C09134=1209.078,130.701,-51.461,-178.311,5.912,148.550
C09135=1209.083,130.452,-51.442,-178.314,5.911,148.551
C09136=1209.088,130.204,-51.422,-178.316,5.909,148.551
C09137=1209.093,129.954,-51.402,-178.318,5.908,148.552
C09138=1209.097,129.705,-51.382,-178.322,5.907,148.552
C09139=1209.102,129.455,-51.362,-178.324,5.906,148.553
C09140=1209.106,129.206,-51.342,-178.327,5.904,148.553
C09141=1209.112,128.957,-51.322,-178.329,5.904,148.554
C09142=1209.117,128.708,-51.301,-178.332,5.902,148.554
C09143=1209.121,128.459,-51.282,-178.334,5.901,148.555
C09144=1209.126,128.210,-51.261,-178.337,5.899,148.555
C09145=1209.131,127.960,-51.242,-178.340,5.899,148.556
C09146=1209.135,127.711,-51.221,-178.342,5.897,148.556
C09147=1209.140,127.462,-51.202,-178.345,5.896,148.557
C09148=1209.145,127.213,-51.182,-178.348,5.895,148.557
C09149=1209.150,126.964,-51.162,-178.350,5.894,148.558
C09150=1209.154,126.715,-51.142,-178.353,5.892,148.558
C09151=1209.159,126.466,-51.122,-178.355,5.891,148.559
C09152=1209.164,126.217,-51.102,-178.358,5.890,148.559
C09153=1209.169,125.968,-51.082,-178.360,5.889,148.560
C09154=1209.173,125.718,-51.063,-178.363,5.888,148.560
C09155=1209.178,125.469,-51.042,-178.366,5.886,148.561
C09156=1209.183,125.220,-51.023,-178.368,5.885,148.561
C09157=1209.188,124.971,-51.003,-178.371,5.884,148.562
C09158=1209.192,124.722,-50.983,-178.373,5.883,148.562
C09159=1209.197,124.472,-50.963,-178.376,5.882,148.563
C09160=1209.202,124.224,-50.943,-178.378,5.881,148.563
C09161=1209.207,123.974,-50.924,-178.381,5.879,148.564
C09162=1209.211,123.725,-50.904,-178.384,5.878,148.564
C09163=1209.216,123.476,-50.884,-178.386,5.877,148.565
C09164=1209.221,123.227,-50.864,-178.389,5.876,148.565
C09165=1209.226,122.977,-50.845,-178.392,5.874,148.566
C09166=1209.231,122.728,-50.825,-178.394,5.874,148.566
C09167=1209.236,122.480,-50.805,-178.396,5.873,148.567
C09168=1209.241,122.230,-50.785,-178.399,5.871,148.567
C09169=1209.245,121.980,-50.766,-178.402,5.870,148.568
C09170=1209.250,121.731,-50.746,-178.405,5.869,148.568
C09171=1209.254,121.483,-50.727,-178.407,5.868,148.569
C09172=1209.259,121.233,-50.707,-178.410,5.866,148.569
C09173=1209.264,120.984,-50.687,-178.412,5.865,148.570
C09174=1209.269,120.735,-50.668,-178.415,5.864,148.570
C09175=1209.274,120.485,-50.648,-178.417,5.863,148.571
C09176=1209.278,120.236,-50.628,-178.420,5.862,148.571
C09177=1209.284,119.988,-50.609,-178.423,5.861,148.572
C09178=1209.288,119.738,-50.589,-178.425,5.860,148.572
C09179=1209.292,119.489,-50.570,-178.428,5.858,148.573
C09180=1209.298,119.240,-50.551,-178.430,5.857,148.573
C09181=1209.303,118.990,-50.531,-178.433,5.856,148.574
C09182=1209.307,118.741,-50.511,-178.436,5.855,148.574
C09183=1209.312,118.492,-50.491,-178.438,5.854,148.575
C09184=1209.317,118.243,-50.472,-178.441,5.853,148.575
C09185=1209.322,117.994,-50.453,-178.443,5.852,148.576
C09186=1209.326,117.745,-50.433,-178.446,5.850,148.576
C09187=1209.331,117.495,-50.414,-178.449,5.850,148.577
C09188=1209.336,117.246,-50.394,-178.451,5.848,148.577
C09189=1209.341,116.997,-50.375,-178.454,5.847,148.578
C09190=1209.345,116.747,-50.356,-178.456,5.846,148.579
C09191=1209.351,116.499,-50.336,-178.459,5.845,148.579
C09192=1209.355,116.249,-50.317,-178.461,5.844,148.580
C09193=1209.361,116.000,-50.297,-178.464,5.842,148.580
C09194=1209.365,115.751,-50.278,-178.467,5.842,148.581
C09195=1209.369,115.501,-50.259,-178.469,5.841,148.581
C09196=1209.375,115.252,-50.239,-178.472,5.839,148.582
C09197=1209.379,115.003,-50.220,-178.474,5.838,148.582
C09198=1209.384,114.754,-50.201,-178.477,5.837,148.583
C09199=1209.389,114.505,-50.181,-178.479,5.836,148.583
C09200=1209.394,114.256,-50.162,-178.482,5.835,148.584
C09201=1209.399,114.006,-50.142,-178.485,5.834,148.584
C09202=1209.403,113.757,-50.123,-178.487,5.833,148.585
C09203=1209.408,113.508,-50.104,-178.490,5.831,148.585
C09204=1209.413,113.259,-50.084,-178.493,5.831,148.586
C09205=1209.418,113.010,-50.066,-178.495,5.830,148.586
C09206=1209.422,112.761,-50.046,-178.498,5.828,148.587
C09207=1209.428,112.512,-50.027,-178.500,5.827,148.587
C09208=1209.432,112.262,-50.008,-178.503,5.826,148.588
C09209=1209.437,112.013,-49.989,-178.505,5.825,148.588
C09210=1209.442,111.763,-49.969,-178.508,5.824,148.589
C09211=1209.446,111.514,-49.950,-178.511,5.822,148.589
C09212=1209.451,111.265,-49.931,-178.513,5.822,148.590
C09213=1209.456,111.016,-49.911,-178.516,5.820,148.590
C09214=1209.461,110.767,-49.893,-178.519,5.820,148.591
C09215=1209.466,110.517,-49.874,-178.521,5.819,148.592
C09216=1209.470,110.268,-49.855,-178.524,5.817,148.592
C09217=1209.475,110.019,-49.835,-178.527,5.817,148.593
C09218=1209.481,109.770,-49.816,-178.529,5.816,148.593
C09219=1209.485,109.521,-49.797,-178.532,5.814,148.594
C09220=1209.490,109.271,-49.779,-178.534,5.813,148.594
C09221=1209.494,109.022,-49.760,-178.537,5.812,148.595
C09222=1209.500,108.773,-49.740,-178.539,5.811,148.595
C09223=1209.504,108.524,-49.721,-178.542,5.810,148.596
C09224=1209.509,108.274,-49.703,-178.545,5.809,148.596
C09225=1209.515,108.025,-49.683,-178.547,5.808,148.597
C09226=1209.519,107.776,-49.664,-178.549,5.807,148.597
C09227=1209.524,107.508,-49.644,-178.553,5.806,148.598
C09228=1209.529,107.239,-49.623,-178.555,5.805,148.599
C09229=1209.534,106.971,-49.604,-178.558,5.803,148.599
C09230=1209.539,106.702,-49.583,-178.561,5.802,148.600
C09231=1209.545,106.453,-49.563,-178.564,5.801,148.600
C09232=1209.549,106.203,-49.545,-178.566,5.800,148.601
C09233=1209.554,105.954,-49.526,-178.569,5.799,148.601
C09234=1209.559,105.706,-49.507,-178.571,5.798,148.602
C09235=1209.564,105.456,-49.488,-178.574,5.797,148.602
C09236=1209.569,105.207,-49.469,-178.576,5.796,148.603
C09237=1209.573,104.957,-49.451,-178.579,5.795,148.603
C09238=1209.578,104.708,-49.432,-178.582,5.794,148.604
C09239=1209.583,104.460,-49.413,-178.584,5.793,148.604
C09240=1209.588,104.210,-49.394,-178.587,5.792,148.605
C09241=1209.592,103.961,-49.375,-178.589,5.791,148.606
C09242=1209.598,103.711,-49.356,-178.592,5.790,148.606
C09243=1209.602,103.462,-49.338,-178.594,5.789,148.607
C09244=1209.608,103.213,-49.319,-178.597,5.788,148.607
C09245=1209.612,102.964,-49.300,-178.600,5.786,148.608
C09246=1209.617,102.714,-49.282,-178.602,5.786,148.608
C09247=1209.621,102.465,-49.263,-178.604,5.785,148.609
C09248=1209.626,102.216,-49.245,-178.608,5.783,148.609
C09249=1209.632,101.967,-49.225,-178.610,5.783,148.610
C09250=1209.636,101.717,-49.207,-178.612,5.782,148.610
C09251=1209.641,101.468,-49.188,-178.616,5.780,148.611
C09252=1209.646,101.219,-49.170,-178.618,5.780,148.611
C09253=1209.650,100.970,-49.151,-178.620,5.779,148.612
C09254=1209.655,100.720,-49.133,-178.623,5.777,148.612
C09255=1209.661,100.472,-49.113,-178.626,5.777,148.613
C09256=1209.665,100.222,-49.095,-178.628,5.776,148.614
C09257=1209.670,99.972,-49.076,-178.631,5.774,148.614
C09258=1209.675,99.724,-49.058,-178.634,5.774,148.615
C09259=1209.679,99.474,-49.039,-178.636,5.773,148.615
C09260=1209.685,99.225,-49.020,-178.639,5.771,148.616
C09261=1209.690,98.976,-49.002,-178.641,5.770,148.616
C09262=1209.694,98.726,-48.984,-178.644,5.770,148.617
C09263=1209.699,98.477,-48.965,-178.646,5.769,148.618
C09264=1209.704,98.228,-48.946,-178.649,5.767,148.618
C09265=1209.709,97.978,-48.928,-178.652,5.767,148.619
C09266=1209.713,97.729,-48.909,-178.654,5.766,148.619
C09267=1209.719,97.480,-48.891,-178.657,5.765,148.620
C09268=1209.723,97.230,-48.872,-178.659,5.764,148.620
C09269=1209.728,96.982,-48.854,-178.662,5.763,148.621
C09270=1209.733,96.732,-48.836,-178.665,5.762,148.621
C09271=1209.738,96.483,-48.817,-178.667,5.761,148.622
C09272=1209.742,96.234,-48.798,-178.670,5.760,148.622
C09273=1209.747,95.984,-48.780,-178.672,5.759,148.623
C09274=1209.752,95.735,-48.762,-178.675,5.758,148.624
C09275=1209.758,95.486,-48.744,-178.677,5.757,148.624
C09276=1209.762,95.236,-48.725,-178.680,5.756,148.625
C09277=1209.767,94.987,-48.707,-178.683,5.755,148.625
C09278=1209.772,94.738,-48.689,-178.685,5.754,148.626
C09279=1209.776,94.489,-48.671,-178.688,5.753,148.626
C09280=1209.782,94.239,-48.652,-178.691,5.752,148.627
C09281=1209.786,93.990,-48.633,-178.693,5.751,148.627
C09282=1209.791,93.741,-48.615,-178.696,5.750,148.628
C09283=1209.796,93.492,-48.597,-178.698,5.749,148.628
C09284=1209.800,93.242,-48.579,-178.701,5.748,148.629
C09285=1209.805,92.993,-48.561,-178.703,5.747,148.630
C09286=1209.811,92.743,-48.542,-178.706,5.746,148.630
C09287=1209.815,92.495,-48.523,-178.708,5.746,148.631
C09288=1209.820,92.245,-48.505,-178.711,5.744,148.631
C09289=1209.825,91.996,-48.487,-178.714,5.744,148.632
C09290=1209.830,91.747,-48.469,-178.716,5.743,148.633
C09291=1209.834,91.497,-48.451,-178.719,5.741,148.633
C09292=1209.839,91.248,-48.433,-178.721,5.741,148.634
C09293=1209.844,90.998,-48.414,-178.724,5.740,148.634
C09294=1209.849,90.749,-48.396,-178.726,5.739,148.635
C09295=1209.854,90.500,-48.378,-178.729,5.738,148.635
C09296=1209.859,90.250,-48.360,-178.732,5.737,148.636
C09297=1209.864,90.001,-48.342,-178.734,5.736,148.636
C09298=1209.869,89.752,-48.324,-178.736,5.735,148.637
C09299=1209.873,89.503,-48.305,-178.739,5.734,148.637
C09300=1209.878,89.254,-48.287,-178.742,5.733,148.638
C09301=1209.883,89.005,-48.269,-178.744,5.732,148.639
C09302=1209.888,88.755,-48.251,-178.747,5.732,148.639
C09303=1209.893,88.506,-48.233,-178.750,5.730,148.640
C09304=1209.898,88.257,-48.215,-178.752,5.729,148.640
C09305=1209.903,88.007,-48.198,-178.755,5.729,148.641
C09306=1209.907,87.757,-48.180,-178.757,5.728,148.641
C09307=1209.912,87.508,-48.162,-178.760,5.727,148.642
C09308=1209.917,87.259,-48.144,-178.763,5.726,148.643
C09309=1209.922,87.010,-48.126,-178.765,5.725,148.643
C09310=1209.927,86.761,-48.108,-178.768,5.724,148.644
C09311=1209.932,86.511,-48.090,-178.771,5.723,148.644
C09312=1209.937,86.262,-48.072,-178.773,5.722,148.645
C09313=1209.941,86.013,-48.054,-178.775,5.722,148.645
C09314=1209.946,85.763,-48.036,-178.778,5.721,148.646
C09315=1209.951,85.514,-48.018,-178.781,5.719,148.646
C09316=1209.956,85.265,-48.000,-178.783,5.719,148.647
C09317=1209.961,85.015,-47.982,-178.786,5.718,148.648
C09318=1209.966,84.766,-47.964,-178.788,5.717,148.648
C09319=1209.971,84.517,-47.946,-178.791,5.717,148.649
C09320=1209.976,84.268,-47.928,-178.794,5.715,148.649
C09321=1209.980,84.018,-47.910,-178.796,5.714,148.650
C09322=1209.985,83.769,-47.892,-178.799,5.714,148.651
C09323=1209.991,83.519,-47.875,-178.801,5.713,148.651
C09324=1209.996,83.270,-47.857,-178.804,5.711,148.652
C09325=1210.000,83.021,-47.839,-178.807,5.711,148.652
C09326=1210.005,82.772,-47.821,-178.809,5.710,148.653
C09327=1210.010,82.522,-47.803,-178.811,5.709,148.653
C09328=1210.014,82.272,-47.786,-178.814,5.709,148.654
C09329=1210.019,82.023,-47.768,-178.817,5.707,148.654
C09330=1210.024,81.774,-47.750,-178.819,5.706,148.655
C09331=1210.029,81.505,-47.732,-178.822,5.706,148.656
C09332=1210.035,81.238,-47.713,-178.825,5.704,148.656
C09333=1210.040,80.969,-47.693,-178.827,5.703,148.657
C09334=1210.046,80.701,-47.674,-178.830,5.703,148.658
C09335=1210.050,80.451,-47.656,-178.833,5.702,148.658
C09336=1210.055,80.202,-47.638,-178.836,5.701,148.659
C09337=1210.061,79.952,-47.621,-178.838,5.700,148.659
C09338=1210.065,79.704,-47.604,-178.841,5.699,148.660
C09339=1210.070,79.454,-47.586,-178.843,5.699,148.661
C09340=1210.075,79.205,-47.569,-178.846,5.697,148.661
C09341=1210.080,78.955,-47.551,-178.849,5.697,148.662
C09342=1210.085,78.706,-47.533,-178.851,5.696,148.662
C09343=1210.089,78.457,-47.516,-178.853,5.695,148.663
C09344=1210.094,78.208,-47.498,-178.856,5.694,148.663
C09345=1210.099,77.958,-47.481,-178.859,5.693,148.664
C09346=1210.104,77.709,-47.463,-178.861,5.692,148.664
C09347=1210.109,77.459,-47.445,-178.864,5.692,148.665
C09348=1210.114,77.210,-47.428,-178.867,5.691,148.666
C09349=1210.118,76.961,-47.410,-178.869,5.690,148.666
C09350=1210.124,76.711,-47.393,-178.872,5.689,148.667
C09351=1210.129,76.462,-47.375,-178.875,5.688,148.668
C09352=1210.133,76.213,-47.357,-178.877,5.687,148.668
C09353=1210.138,75.963,-47.340,-178.879,5.687,148.669
C09354=1210.143,75.714,-47.322,-178.882,5.686,148.669
C09355=1210.148,75.464,-47.305,-178.884,5.685,148.670
C09356=1210.152,75.215,-47.288,-178.887,5.684,148.670
C09357=1210.158,74.966,-47.271,-178.890,5.683,148.671
C09358=1210.163,74.717,-47.253,-178.892,5.682,148.671
C09359=1210.168,74.468,-47.236,-178.895,5.682,148.672
C09360=1210.172,74.218,-47.218,-178.897,5.681,148.673
C09361=1210.178,73.969,-47.201,-178.900,5.681,148.673
C09362=1210.182,73.719,-47.184,-178.903,5.679,148.674
C09363=1210.187,73.470,-47.166,-178.905,5.678,148.674
C09364=1210.192,73.220,-47.149,-178.908,5.678,148.675
C09365=1210.196,72.971,-47.131,-178.910,5.677,148.676
C09366=1210.202,72.721,-47.114,-178.913,5.676,148.676
C09367=1210.207,72.472,-47.096,-178.915,5.676,148.677
C09368=1210.212,72.224,-47.080,-178.918,5.674,148.677
C09369=1210.217,71.974,-47.063,-178.921,5.673,148.678
C09370=1210.222,71.725,-47.045,-178.923,5.673,148.679
C09371=1210.226,71.475,-47.028,-178.925,5.672,148.679
C09372=1210.231,71.226,-47.010,-178.928,5.671,148.680
C09373=1210.236,70.976,-46.993,-178.931,5.671,148.680
C09374=1210.241,70.727,-46.976,-178.934,5.669,148.681
C09375=1210.246,70.478,-46.958,-178.936,5.668,148.681
C09376=1210.251,70.229,-46.942,-178.939,5.668,148.682
C09377=1210.256,69.979,-46.925,-178.941,5.667,148.683
C09378=1210.260,69.730,-46.907,-178.943,5.666,148.683
C09379=1210.265,69.480,-46.890,-178.946,5.666,148.684
C09380=1210.271,69.230,-46.873,-178.949,5.665,148.685
C09381=1210.275,68.981,-46.856,-178.952,5.664,148.685
C09382=1210.281,68.732,-46.838,-178.954,5.663,148.686
C09383=1210.285,68.483,-46.822,-178.957,5.662,148.686
C09384=1210.290,68.233,-46.804,-178.959,5.662,148.687
C09385=1210.295,67.984,-46.787,-178.961,5.661,148.687
C09386=1210.300,67.735,-46.770,-178.964,5.660,148.688
C09387=1210.305,67.486,-46.753,-178.967,5.660,148.689
C09388=1210.310,67.236,-46.736,-178.970,5.658,148.689
C09389=1210.315,66.986,-46.720,-178.972,5.657,148.690
C09390=1210.319,66.737,-46.702,-178.975,5.657,148.690
C09391=1210.324,66.488,-46.685,-178.977,5.656,148.691
C09392=1210.330,66.239,-46.668,-178.979,5.655,148.692
C09393=1210.334,65.989,-46.651,-178.982,5.655,148.692
C09394=1210.339,65.739,-46.634,-178.985,5.654,148.693
C09395=1210.344,65.491,-46.617,-178.987,5.654,148.694
C09396=1210.349,65.241,-46.599,-178.990,5.652,148.694
C09397=1210.354,64.992,-46.583,-178.993,5.651,148.695
C09398=1210.359,64.742,-46.566,-178.995,5.651,148.695
C09399=1210.364,64.493,-46.549,-178.997,5.650,148.696
C09400=1210.369,64.243,-46.532,-179.000,5.649,148.696
C09401=1210.374,63.994,-46.516,-179.003,5.649,148.697
C09402=1210.378,63.745,-46.499,-179.005,5.648,148.698
C09403=1210.383,63.495,-46.481,-179.007,5.647,148.698
C09404=1210.388,63.246,-46.464,-179.011,5.646,148.699
C09405=1210.394,62.997,-46.447,-179.013,5.645,148.699
C09406=1210.398,62.747,-46.431,-179.016,5.645,148.700
C09407=1210.403,62.498,-46.414,-179.018,5.644,148.701
C09408=1210.408,62.248,-46.397,-179.021,5.643,148.701
C09409=1210.413,61.999,-46.380,-179.023,5.643,148.702
C09410=1210.418,61.750,-46.363,-179.026,5.642,148.703
C09411=1210.423,61.500,-46.347,-179.028,5.641,148.703
C09412=1210.428,61.251,-46.330,-179.031,5.641,148.704
C09413=1210.433,61.001,-46.313,-179.034,5.639,148.704
C09414=1210.437,60.752,-46.296,-179.036,5.639,148.705
C09415=1210.442,60.503,-46.280,-179.039,5.638,148.705
C09416=1210.448,60.253,-46.263,-179.041,5.637,148.706
C09417=1210.452,60.004,-46.246,-179.044,5.637,148.707
C09418=1210.457,59.754,-46.229,-179.046,5.636,148.707
C09419=1210.462,59.505,-46.213,-179.049,5.635,148.708
C09420=1210.467,59.256,-46.196,-179.051,5.635,148.709
C09421=1210.471,59.006,-46.179,-179.054,5.634,148.709
C09422=1210.477,58.757,-46.162,-179.056,5.633,148.710
C09423=1210.482,58.508,-46.146,-179.059,5.633,148.710
C09424=1210.486,58.258,-46.129,-179.062,5.631,148.711
C09425=1210.492,58.009,-46.113,-179.065,5.631,148.712
C09426=1210.497,57.759,-46.096,-179.067,5.630,148.712
C09427=1210.501,57.510,-46.079,-179.069,5.629,148.713
C09428=1210.506,57.261,-46.063,-179.072,5.629,148.713
C09429=1210.512,57.011,-46.046,-179.075,5.628,148.714
C09430=1210.516,56.762,-46.029,-179.077,5.627,148.714
C09431=1210.521,56.513,-46.013,-179.079,5.627,148.715
C09432=1210.527,56.262,-45.996,-179.082,5.626,148.716
C09433=1210.532,56.014,-45.980,-179.085,5.626,148.716
C09434=1210.536,55.764,-45.963,-179.087,5.625,148.717
C09435=1210.541,55.496,-45.946,-179.090,5.623,148.718
C09436=1210.547,55.227,-45.928,-179.093,5.623,148.718
C09437=1210.552,54.959,-45.910,-179.095,5.622,148.719
C09438=1210.557,54.690,-45.892,-179.098,5.622,148.720
C09439=1210.562,54.441,-45.876,-179.101,5.621,148.720
C09440=1210.568,54.191,-45.859,-179.103,5.621,148.721
C09441=1210.573,53.942,-45.843,-179.106,5.620,148.722
C09442=1210.577,53.693,-45.826,-179.109,5.618,148.722
C09443=1210.582,53.443,-45.810,-179.111,5.618,148.723
C09444=1210.587,53.194,-45.794,-179.114,5.617,148.723
C09445=1210.592,52.945,-45.777,-179.117,5.617,148.724
C09446=1210.597,52.695,-45.760,-179.119,5.616,148.725
C09447=1210.602,52.445,-45.744,-179.121,5.615,148.725
C09448=1210.607,52.196,-45.728,-179.124,5.615,148.726
C09449=1210.612,51.947,-45.711,-179.127,5.614,148.726
C09450=1210.617,51.697,-45.695,-179.129,5.614,148.727
C09451=1210.622,51.448,-45.679,-179.131,5.613,148.728
C09452=1210.626,51.199,-45.662,-179.134,5.612,148.728
C09453=1210.632,50.949,-45.646,-179.137,5.612,148.729
C09454=1210.637,50.699,-45.629,-179.139,5.611,148.730
C09455=1210.642,50.451,-45.613,-179.141,5.610,148.730
C09456=1210.647,50.201,-45.597,-179.144,5.610,148.731
C09457=1210.651,49.951,-45.581,-179.147,5.609,148.731
C09458=1210.656,49.702,-45.564,-179.149,5.609,148.732
C09459=1210.661,49.452,-45.548,-179.152,5.608,148.733
C09460=1210.666,49.203,-45.532,-179.154,5.607,148.733
C09461=1210.671,48.953,-45.516,-179.157,5.607,148.734
C09462=1210.676,48.705,-45.500,-179.160,5.605,148.734
C09463=1210.680,48.455,-45.483,-179.163,5.605,148.735
C09464=1210.686,48.206,-45.467,-179.165,5.604,148.736
C09465=1210.691,47.956,-45.450,-179.167,5.603,148.736
C09466=1210.696,47.706,-45.435,-179.170,5.603,148.737
C09467=1210.701,47.457,-45.418,-179.173,5.602,148.738
C09468=1210.706,47.208,-45.402,-179.175,5.602,148.738
C09469=1210.711,46.958,-45.386,-179.177,5.601,148.739
C09470=1210.716,46.709,-45.370,-179.180,5.600,148.739
C09471=1210.721,46.459,-45.353,-179.183,5.600,148.740
C09472=1210.726,46.210,-45.338,-179.185,5.599,148.741
C09473=1210.730,45.960,-45.321,-179.188,5.599,148.741
C09474=1210.736,45.711,-45.306,-179.190,5.598,148.742
C09475=1210.741,45.462,-45.289,-179.193,5.597,148.743
C09476=1210.746,45.212,-45.273,-179.195,5.597,148.743
C09477=1210.751,44.963,-45.257,-179.198,5.596,148.744
C09478=1210.756,44.713,-45.241,-179.201,5.595,148.745
C09479=1210.761,44.464,-45.225,-179.203,5.595,148.745
C09480=1210.765,44.214,-45.209,-179.205,5.594,148.746
C09481=1210.770,43.965,-45.194,-179.208,5.593,148.746
C09482=1210.775,43.716,-45.177,-179.211,5.593,148.747
C09483=1210.780,43.466,-45.162,-179.213,5.592,148.748
C09484=1210.785,43.218,-45.145,-179.216,5.591,148.748
C09485=1210.790,42.967,-45.129,-179.218,5.591,148.749
C09486=1210.795,42.718,-45.114,-179.221,5.590,148.749
C09487=1210.800,42.469,-45.097,-179.223,5.590,148.750
C09488=1210.805,42.219,-45.081,-179.226,5.589,148.751
C09489=1210.810,41.969,-45.065,-179.228,5.588,148.751
C09490=1210.815,41.720,-45.049,-179.231,5.588,148.752
C09491=1210.820,41.471,-45.034,-179.234,5.587,148.753
C09492=1210.825,41.221,-45.018,-179.236,5.587,148.753
C09493=1210.830,40.972,-45.001,-179.239,5.586,148.754
C09494=1210.835,40.723,-44.986,-179.241,5.585,148.754
C09495=1210.840,40.473,-44.970,-179.244,5.585,148.755
C09496=1210.845,40.224,-44.954,-179.246,5.584,148.756
C09497=1210.849,39.974,-44.938,-179.249,5.584,148.756
C09498=1210.855,39.724,-44.923,-179.252,5.583,148.757
C09499=1210.860,39.475,-44.907,-179.254,5.583,148.758
C09500=1210.865,39.226,-44.890,-179.256,5.582,148.758
C09501=1210.869,38.976,-44.875,-179.259,5.581,148.759
C09502=1210.875,38.727,-44.860,-179.262,5.581,148.760
C09503=1210.880,38.477,-44.844,-179.264,5.580,148.760
C09504=1210.885,38.228,-44.827,-179.267,5.580,148.761
C09505=1210.890,37.979,-44.812,-179.269,5.579,148.761
C09506=1210.895,37.729,-44.796,-179.272,5.578,148.762
C09507=1210.899,37.480,-44.781,-179.274,5.578,148.763
C09508=1210.905,37.230,-44.765,-179.277,5.577,148.763
C09509=1210.909,36.981,-44.749,-179.280,5.577,148.764
C09510=1210.915,36.731,-44.733,-179.282,5.576,148.765
C09511=1210.919,36.482,-44.718,-179.284,5.575,148.765
C09512=1210.924,36.232,-44.702,-179.287,5.575,148.766
C09513=1210.930,35.983,-44.687,-179.290,5.574,148.767
C09514=1210.935,35.733,-44.671,-179.292,5.573,148.767
C09515=1210.939,35.484,-44.654,-179.295,5.573,148.768
C09516=1210.944,35.235,-44.639,-179.297,5.572,148.768
C09517=1210.949,34.985,-44.624,-179.300,5.572,148.769
C09518=1210.954,34.735,-44.608,-179.302,5.571,148.770
C09519=1210.960,34.486,-44.592,-179.305,5.570,148.770
C09520=1210.964,34.237,-44.577,-179.308,5.570,148.771
C09521=1210.970,33.987,-44.562,-179.310,5.569,148.772
C09522=1210.974,33.737,-44.546,-179.312,5.568,148.772
C09523=1210.979,33.488,-44.531,-179.315,5.568,148.773
C09524=1210.984,33.239,-44.515,-179.318,5.567,148.773
C09525=1210.989,32.989,-44.499,-179.320,5.568,148.774
C09526=1210.994,32.740,-44.484,-179.322,5.567,148.775
C09527=1210.999,32.490,-44.469,-179.325,5.567,148.776
C09528=1211.005,32.241,-44.453,-179.327,5.566,148.776
C09529=1211.009,31.991,-44.438,-179.330,5.565,148.777
C09530=1211.014,31.742,-44.422,-179.333,5.565,148.777
C09531=1211.019,31.492,-44.406,-179.335,5.564,148.778
C09532=1211.024,31.243,-44.391,-179.338,5.564,148.779
C09533=1211.029,30.993,-44.375,-179.341,5.563,148.779
C09534=1211.034,30.744,-44.360,-179.343,5.562,148.780
C09535=1211.039,30.494,-44.345,-179.345,5.562,148.780
C09536=1211.044,30.245,-44.329,-179.348,5.561,148.781
C09537=1211.049,29.995,-44.313,-179.351,5.561,148.782
C09538=1211.054,29.746,-44.298,-179.353,5.560,148.783
C09539=1211.059,29.477,-44.281,-179.356,5.560,148.783
C09540=1211.065,29.208,-44.265,-179.359,5.559,148.784
C09541=1211.070,28.940,-44.249,-179.361,5.558,148.785
C09542=1211.076,28.672,-44.232,-179.364,5.558,148.785
C09543=1211.080,28.423,-44.217,-179.366,5.557,148.786
C09544=1211.086,28.173,-44.202,-179.369,5.557,148.787
C09545=1211.091,27.922,-44.186,-179.372,5.556,148.787
C09546=1211.095,27.673,-44.171,-179.374,5.555,148.788
C09547=1211.101,27.424,-44.155,-179.377,5.555,148.788
C09548=1211.105,27.175,-44.140,-179.379,5.554,148.789
C09549=1211.111,26.925,-44.125,-179.382,5.554,148.790
C09550=1211.115,26.676,-44.109,-179.384,5.553,148.790
C09551=1211.120,26.426,-44.094,-179.387,5.553,148.791
C09552=1211.126,26.176,-44.079,-179.389,5.552,148.792
C09553=1211.131,25.927,-44.064,-179.392,5.551,148.792
C09554=1211.136,25.678,-44.048,-179.394,5.552,148.793
C09555=1211.141,25.429,-44.033,-179.397,5.551,148.794
C09556=1211.146,25.178,-44.018,-179.399,5.551,148.794
C09557=1211.150,24.929,-44.003,-179.402,5.550,148.795
C09558=1211.156,24.679,-43.987,-179.405,5.550,148.796
C09559=1211.160,24.430,-43.972,-179.407,5.549,148.796
C09560=1211.166,24.180,-43.958,-179.409,5.548,148.797
C09561=1211.171,23.931,-43.943,-179.412,5.548,148.797
C09562=1211.176,23.682,-43.927,-179.415,5.547,148.798
C09563=1211.181,23.433,-43.912,-179.417,5.547,148.799
C09564=1211.186,23.182,-43.897,-179.420,5.546,148.799
C09565=1211.190,22.933,-43.882,-179.423,5.546,148.800
C09566=1211.195,22.684,-43.867,-179.424,5.545,148.801
C09567=1211.200,22.434,-43.851,-179.427,5.545,148.801
C09568=1211.205,22.185,-43.837,-179.429,5.544,148.802
C09569=1211.211,21.935,-43.821,-179.432,5.544,148.803
C09570=1211.215,21.686,-43.806,-179.435,5.543,148.803
C09571=1211.221,21.436,-43.791,-179.437,5.543,148.804
C09572=1211.226,21.187,-43.776,-179.440,5.542,148.805
C09573=1211.230,20.937,-43.761,-179.442,5.541,148.805
C09574=1211.236,20.687,-43.746,-179.445,5.541,148.806
C09575=1211.240,20.438,-43.731,-179.448,5.540,148.806
C09576=1211.246,20.188,-43.716,-179.450,5.540,148.807
C09577=1211.251,19.939,-43.701,-179.452,5.540,148.808
C09578=1211.255,19.690,-43.686,-179.455,5.540,148.809
C09579=1211.261,19.440,-43.671,-179.458,5.539,148.809
C09580=1211.266,19.191,-43.656,-179.460,5.538,148.810
C09581=1211.271,18.941,-43.642,-179.462,5.538,148.810
C09582=1211.276,18.692,-43.627,-179.465,5.537,148.811
C09583=1211.281,18.443,-43.612,-179.468,5.537,148.812
C09584=1211.286,18.193,-43.597,-179.470,5.536,148.812
C09585=1211.291,17.944,-43.582,-179.473,5.536,148.813
C09586=1211.296,17.694,-43.567,-179.476,5.535,148.814
C09587=1211.301,17.444,-43.552,-179.478,5.535,148.814
C09588=1211.306,17.195,-43.538,-179.480,5.534,148.815
C09589=1211.311,16.946,-43.523,-179.482,5.534,148.816
C09590=1211.317,16.696,-43.508,-179.485,5.533,148.816
C09591=1211.321,16.447,-43.493,-179.488,5.533,148.817
C09592=1211.326,16.197,-43.478,-179.490,5.532,148.818
C09593=1211.332,15.947,-43.463,-179.493,5.532,148.818
C09594=1211.336,15.698,-43.449,-179.496,5.531,148.819
C09595=1211.341,15.449,-43.434,-179.498,5.532,148.820
C09596=1211.346,15.199,-43.419,-179.500,5.531,148.820
C09597=1211.351,14.949,-43.404,-179.503,5.530,148.821
C09598=1211.356,14.700,-43.389,-179.505,5.530,148.822
C09599=1211.361,14.451,-43.374,-179.508,5.529,148.822
C09600=1211.366,14.201,-43.360,-179.511,5.529,148.823
C09601=1211.372,13.951,-43.345,-179.513,5.528,148.824
C09602=1211.376,13.702,-43.330,-179.516,5.528,148.824
C09603=1211.381,13.452,-43.316,-179.518,5.528,148.825
C09604=1211.386,13.203,-43.301,-179.520,5.527,148.825
C09605=1211.392,12.953,-43.286,-179.523,5.527,148.826
C09606=1211.397,12.703,-43.272,-179.525,5.526,148.827
C09607=1211.401,12.454,-43.257,-179.528,5.526,148.827
C09608=1211.406,12.205,-43.243,-179.531,5.525,148.828
C09609=1211.412,11.955,-43.227,-179.533,5.525,148.829
C09610=1211.417,11.705,-43.213,-179.536,5.524,148.829
C09611=1211.422,11.456,-43.198,-179.538,5.524,148.830
C09612=1211.426,11.207,-43.184,-179.540,5.523,148.831
C09613=1211.431,10.957,-43.169,-179.543,5.523,148.831
C09614=1211.437,10.707,-43.154,-179.545,5.522,148.832
C09615=1211.441,10.458,-43.139,-179.548,5.522,148.833
C09616=1211.446,10.208,-43.125,-179.551,5.521,148.833
C09617=1211.451,9.958,-43.111,-179.553,5.521,148.834
C09618=1211.456,9.709,-43.097,-179.556,5.521,148.835
C09619=1211.462,9.460,-43.082,-179.558,5.521,148.835
C09620=1211.467,9.210,-43.067,-179.560,5.520,148.836
C09621=1211.472,8.961,-43.053,-179.563,5.519,148.837
C09622=1211.477,8.711,-43.038,-179.566,5.519,148.837
C09623=1211.482,8.462,-43.023,-179.568,5.518,148.838
C09624=1211.487,8.212,-43.009,-179.571,5.518,148.839
C09625=1211.492,7.962,-42.995,-179.573,5.518,148.839
C09626=1211.497,7.713,-42.981,-179.576,5.517,148.840
C09627=1211.501,7.463,-42.966,-179.578,5.517,148.841
C09628=1211.506,7.214,-42.951,-179.581,5.516,148.841
C09629=1211.513,6.964,-42.937,-179.583,5.516,148.842
C09630=1211.518,6.715,-42.923,-179.586,5.515,148.843
C09631=1211.522,6.465,-42.908,-179.588,5.515,148.843
C09632=1211.527,6.216,-42.893,-179.590,5.515,148.844
C09633=1211.532,5.966,-42.879,-179.593,5.514,148.845
C09634=1211.537,5.717,-42.865,-179.596,5.514,148.845
C09635=1211.542,5.467,-42.850,-179.598,5.513,148.846
C09636=1211.548,5.218,-42.837,-179.601,5.513,148.847
C09637=1211.553,4.968,-42.822,-179.604,5.512,148.847
C09638=1211.557,4.718,-42.808,-179.605,5.512,148.848
C09639=1211.562,4.469,-42.793,-179.608,5.512,148.848
C09640=1211.567,4.220,-42.779,-179.611,5.511,148.849
C09641=1211.572,3.970,-42.764,-179.613,5.511,148.850
C09642=1211.578,3.721,-42.751,-179.616,5.510,148.851
C09643=1211.583,3.451,-42.736,-179.619,5.510,148.851
C09644=1211.589,3.182,-42.719,-179.621,5.509,148.852
C09645=1211.594,2.913,-42.704,-179.624,5.509,148.853
C09646=1211.599,2.644,-42.689,-179.627,5.509,148.854
C09647=1211.604,2.394,-42.674,-179.629,5.508,148.854
C09648=1211.609,2.145,-42.660,-179.631,5.508,148.855
C09649=1211.615,1.896,-42.646,-179.634,5.507,148.855
C09650=1211.620,1.646,-42.632,-179.637,5.507,148.856
C09651=1211.625,1.396,-42.618,-179.639,5.506,148.857
C09652=1211.630,1.147,-42.603,-179.641,5.507,148.857
C09653=1211.635,0.898,-42.589,-179.644,5.506,148.858
C09654=1211.640,0.648,-42.575,-179.647,5.506,148.859
C09655=1211.645,0.398,-42.561,-179.649,5.505,148.859
C09656=1211.649,0.149,-42.547,-179.652,5.505,148.860
C09657=1211.654,-0.101,-42.533,-179.654,5.504,148.861
C09658=1211.660,-0.350,-42.519,-179.656,5.504,148.861
C09659=1211.665,-0.600,-42.505,-179.659,5.504,148.862
C09660=1211.670,-0.849,-42.490,-179.661,5.503,148.863
C09661=1211.675,-1.099,-42.476,-179.664,5.503,148.863
C09662=1211.680,-1.348,-42.462,-179.667,5.502,148.864
C09663=1211.685,-1.598,-42.448,-179.669,5.502,148.865
C09664=1211.690,-1.848,-42.434,-179.671,5.502,148.865
C09665=1211.695,-2.097,-42.419,-179.674,5.501,148.866
C09666=1211.701,-2.346,-42.405,-179.677,5.501,148.867
C09667=1211.705,-2.596,-42.392,-179.679,5.500,148.867
C09668=1211.710,-2.846,-42.378,-179.681,5.500,148.868
C09669=1211.715,-3.096,-42.364,-179.684,5.500,148.869
C09670=1211.721,-3.345,-42.350,-179.686,5.499,148.869
C09671=1211.726,-3.594,-42.336,-179.689,5.499,148.870
C09672=1211.731,-3.844,-42.321,-179.692,5.498,148.871
C09673=1211.736,-4.093,-42.308,-179.694,5.499,148.871
C09674=1211.741,-4.343,-42.295,-179.696,5.498,148.872
C09675=1211.746,-4.593,-42.280,-179.699,5.498,148.873
C09676=1211.751,-4.843,-42.266,-179.702,5.497,148.874
C09677=1211.756,-5.092,-42.252,-179.704,5.496,148.874
C09678=1211.761,-5.341,-42.238,-179.706,5.497,148.875
C09679=1211.766,-5.591,-42.224,-179.709,5.496,148.875
C09680=1211.771,-5.840,-42.211,-179.711,5.496,148.876
C09681=1211.776,-6.090,-42.197,-179.714,5.495,148.877
C09682=1211.781,-6.340,-42.182,-179.717,5.495,148.877
C09683=1211.787,-6.589,-42.169,-179.719,5.495,148.878
C09684=1211.792,-6.839,-42.155,-179.721,5.494,148.879
C09685=1211.796,-7.088,-42.141,-179.724,5.494,148.879
C09686=1211.802,-7.337,-42.127,-179.727,5.493,148.880
C09687=1211.807,-7.587,-42.113,-179.729,5.493,148.881
C09688=1211.812,-7.838,-42.100,-179.731,5.493,148.881
C09689=1211.817,-8.086,-42.086,-179.733,5.492,148.882
C09690=1211.822,-8.336,-42.072,-179.736,5.492,148.883
C09691=1211.827,-8.586,-42.058,-179.739,5.491,148.883
C09692=1211.833,-8.835,-42.044,-179.741,5.492,148.884
C09693=1211.837,-9.085,-42.031,-179.744,5.491,148.885
C09694=1211.842,-9.334,-42.016,-179.746,5.491,148.885
C09695=1211.848,-9.584,-42.003,-179.749,5.490,148.886
C09696=1211.853,-9.834,-41.989,-179.752,5.490,148.887
C09697=1211.857,-10.083,-41.975,-179.754,5.490,148.888
C09698=1211.863,-10.333,-41.962,-179.756,5.489,148.888
C09699=1211.868,-10.582,-41.948,-179.758,5.489,148.889
C09700=1211.872,-10.831,-41.935,-179.761,5.488,148.889
C09701=1211.878,-11.081,-41.921,-179.763,5.488,148.890
C09702=1211.883,-11.331,-41.907,-179.766,5.488,148.891
C09703=1211.888,-11.581,-41.894,-179.768,5.487,148.891
C09704=1211.893,-11.830,-41.880,-179.771,5.487,148.892
C09705=1211.898,-12.079,-41.866,-179.773,5.487,148.893
C09706=1211.903,-12.329,-41.853,-179.776,5.487,148.894
C09707=1211.908,-12.579,-41.839,-179.778,5.486,148.894
C09708=1211.914,-12.829,-41.825,-179.781,5.486,148.895
C09709=1211.918,-13.078,-41.812,-179.784,5.485,148.896
C09710=1211.923,-13.327,-41.798,-179.786,5.486,148.896
C09711=1211.929,-13.577,-41.784,-179.788,5.485,148.897
C09712=1211.933,-13.827,-41.771,-179.791,5.484,148.897
C09713=1211.939,-14.076,-41.757,-179.793,5.484,148.898
C09714=1211.944,-14.326,-41.743,-179.795,5.484,148.899
C09715=1211.949,-14.575,-41.731,-179.798,5.484,148.900
C09716=1211.954,-14.825,-41.716,-179.801,5.483,148.900
C09717=1211.959,-15.074,-41.704,-179.803,5.483,148.901
C09718=1211.964,-15.324,-41.689,-179.805,5.483,148.902
C09719=1211.970,-15.574,-41.676,-179.808,5.482,148.902
C09720=1211.974,-15.823,-41.663,-179.811,5.482,148.903
C09721=1211.979,-16.073,-41.649,-179.813,5.481,148.904
C09722=1211.984,-16.322,-41.636,-179.816,5.482,148.904
C09723=1211.989,-16.573,-41.622,-179.818,5.481,148.905
C09724=1211.994,-16.821,-41.609,-179.820,5.480,148.906
C09725=1211.999,-17.072,-41.595,-179.823,5.480,148.906
C09726=1212.005,-17.321,-41.582,-179.825,5.480,148.907
C09727=1212.009,-17.571,-41.568,-179.828,5.480,148.908
C09728=1212.015,-17.820,-41.555,-179.830,5.479,148.908
C09729=1212.019,-18.070,-41.541,-179.833,5.479,148.909
C09730=1212.025,-18.319,-41.528,-179.835,5.479,148.910
C09731=1212.030,-18.569,-41.515,-179.838,5.479,148.910
C09732=1212.035,-18.818,-41.501,-179.840,5.478,148.911
C09733=1212.040,-19.068,-41.488,-179.843,5.478,148.912
C09734=1212.046,-19.317,-41.475,-179.845,5.478,148.913
C09735=1212.050,-19.567,-41.462,-179.847,5.477,148.913
C09736=1212.056,-19.817,-41.448,-179.850,5.477,148.914
C09737=1212.060,-20.066,-41.435,-179.853,5.476,148.914
C09738=1212.066,-20.316,-41.421,-179.855,5.476,148.915
C09739=1212.070,-20.566,-41.408,-179.857,5.476,148.916
C09740=1212.076,-20.815,-41.395,-179.860,5.475,148.916
C09741=1212.081,-21.064,-41.382,-179.862,5.476,148.917
C09742=1212.086,-21.315,-41.368,-179.865,5.475,148.918
C09743=1212.091,-21.563,-41.355,-179.867,5.475,148.919
C09744=1212.097,-21.814,-41.342,-179.870,5.474,148.919
C09745=1212.102,-22.063,-41.329,-179.872,5.475,148.920
C09746=1212.107,-22.313,-41.315,-179.875,5.474,148.921
C09747=1212.112,-22.582,-41.301,-179.878,5.474,148.921
C09748=1212.118,-22.852,-41.287,-179.880,5.473,148.922
C09749=1212.123,-23.121,-41.272,-179.883,5.473,148.923
C09750=1212.128,-23.391,-41.258,-179.886,5.472,148.923
C09751=1212.134,-23.641,-41.245,-179.888,5.472,148.924
C09752=1212.139,-23.889,-41.232,-179.890,5.472,148.925
C09753=1212.144,-24.139,-41.219,-179.893,5.472,148.926
C09754=1212.149,-24.389,-41.206,-179.895,5.472,148.926
C09755=1212.154,-24.639,-41.193,-179.898,5.471,148.927
C09756=1212.160,-24.888,-41.179,-179.900,5.471,148.928
C09757=1212.164,-25.138,-41.166,-179.903,5.470,148.928
C09758=1212.169,-25.387,-41.153,-179.905,5.471,148.929
C09759=1212.175,-25.637,-41.140,-179.907,5.470,148.929
C09760=1212.180,-25.887,-41.127,-179.910,5.469,148.930
C09761=1212.185,-26.136,-41.115,-179.912,5.470,148.931
C09762=1212.190,-26.386,-41.100,-179.915,5.469,148.932
C09763=1212.195,-26.635,-41.088,-179.917,5.469,148.932
C09764=1212.201,-26.885,-41.074,-179.920,5.468,148.933
C09765=1212.205,-27.135,-41.061,-179.922,5.469,148.934
C09766=1212.210,-27.384,-41.049,-179.925,5.468,148.934
C09767=1212.216,-27.634,-41.036,-179.927,5.468,148.935
C09768=1212.221,-27.884,-41.023,-179.929,5.468,148.936
C09769=1212.225,-28.133,-41.009,-179.932,5.467,148.936
C09770=1212.230,-28.383,-40.996,-179.935,5.467,148.937
C09771=1212.236,-28.632,-40.983,-179.937,5.466,148.938
C09772=1212.241,-28.881,-40.971,-179.939,5.466,148.938
C09773=1212.245,-29.132,-40.958,-179.942,5.466,148.939
C09774=1212.251,-29.381,-40.944,-179.944,5.465,148.940
C09775=1212.256,-29.630,-40.932,-179.946,5.466,148.940
C09776=1212.261,-29.880,-40.919,-179.949,5.465,148.941
C09777=1212.267,-30.130,-40.906,-179.952,5.465,148.942
C09778=1212.272,-30.379,-40.893,-179.954,5.465,148.942
C09779=1212.277,-30.629,-40.880,-179.956,5.465,148.943
C09780=1212.282,-30.879,-40.868,-179.959,5.464,148.944
C09781=1212.287,-31.128,-40.854,-179.962,5.464,148.945
C09782=1212.292,-31.378,-40.841,-179.964,5.464,148.945
C09783=1212.297,-31.628,-40.829,-179.967,5.464,148.946
C09784=1212.302,-31.877,-40.816,-179.969,5.463,148.946
C09785=1212.308,-32.127,-40.803,-179.971,5.463,148.947
C09786=1212.313,-32.377,-40.790,-179.973,5.463,148.948
C09787=1212.318,-32.626,-40.777,-179.976,5.462,148.949
C09788=1212.322,-32.876,-40.764,-179.978,5.462,148.949
C09789=1212.327,-33.125,-40.752,-179.981,5.462,148.950
C09790=1212.333,-33.375,-40.739,-179.984,5.461,148.951
C09791=1212.338,-33.624,-40.726,-179.986,5.462,148.951
C09792=1212.343,-33.874,-40.713,-179.988,5.461,148.952
C09793=1212.348,-34.124,-40.700,-179.991,5.461,148.953
C09794=1212.353,-34.373,-40.688,-179.993,5.461,148.953
C09795=1212.358,-34.623,-40.674,-179.996,5.461,148.954
C09796=1212.364,-34.873,-40.662,-179.998,5.460,148.955
C09797=1212.369,-35.123,-40.650,179.999,5.459,148.955
C09798=1212.374,-35.372,-40.637,179.997,5.460,148.956
C09799=1212.379,-35.622,-40.624,179.995,5.459,148.957
C09800=1212.384,-35.872,-40.611,179.992,5.459,148.957
C09801=1212.390,-36.121,-40.598,179.990,5.459,148.958
C09802=1212.395,-36.370,-40.586,179.987,5.459,148.959
C09803=1212.399,-36.620,-40.573,179.985,5.458,148.959
C09804=1212.404,-36.869,-40.560,179.983,5.458,148.960
C09805=1212.410,-37.119,-40.548,179.980,5.458,148.961
C09806=1212.415,-37.369,-40.536,179.977,5.458,148.962
C09807=1212.421,-37.618,-40.523,179.975,5.458,148.962
C09808=1212.425,-37.868,-40.510,179.973,5.457,148.963
C09809=1212.430,-38.118,-40.497,179.970,5.457,148.964
C09810=1212.436,-38.368,-40.485,179.968,5.457,148.964
C09811=1212.441,-38.617,-40.473,179.966,5.456,148.965
C09812=1212.446,-38.867,-40.460,179.963,5.456,148.966
C09813=1212.451,-39.116,-40.447,179.961,5.456,148.966
C09814=1212.456,-39.366,-40.434,179.958,5.456,148.967
C09815=1212.461,-39.616,-40.423,179.956,5.455,148.968
C09816=1212.466,-39.865,-40.410,179.953,5.456,148.968
C09817=1212.471,-40.115,-40.397,179.951,5.455,148.969
C09818=1212.477,-40.364,-40.384,179.948,5.455,148.970
C09819=1212.482,-40.614,-40.372,179.946,5.455,148.970
C09820=1212.487,-40.864,-40.359,179.943,5.455,148.971
C09821=1212.492,-41.113,-40.347,179.941,5.454,148.972
C09822=1212.497,-41.364,-40.334,179.939,5.454,148.973
C09823=1212.502,-41.613,-40.322,179.936,5.454,148.973
C09824=1212.507,-41.862,-40.309,179.934,5.453,148.974
C09825=1212.513,-42.112,-40.297,179.932,5.453,148.974
C09826=1212.518,-42.362,-40.285,179.929,5.453,148.975
C09827=1212.523,-42.611,-40.272,179.926,5.452,148.976
C09828=1212.528,-42.861,-40.259,179.924,5.453,148.977
C09829=1212.533,-43.111,-40.247,179.922,5.452,148.977
C09830=1212.538,-43.360,-40.235,179.919,5.452,148.978
C09831=1212.543,-43.609,-40.222,179.917,5.452,148.979
C09832=1212.549,-43.859,-40.210,179.914,5.452,148.979
C09833=1212.554,-44.109,-40.198,179.912,5.451,148.980
C09834=1212.559,-44.359,-40.186,179.909,5.452,148.981
C09835=1212.564,-44.609,-40.173,179.907,5.451,148.981
C09836=1212.569,-44.858,-40.160,179.905,5.451,148.982
C09837=1212.574,-45.108,-40.148,179.903,5.451,148.983
C09838=1212.580,-45.357,-40.136,179.900,5.450,148.983
C09839=1212.585,-45.607,-40.124,179.898,5.451,148.984
C09840=1212.590,-45.857,-40.111,179.895,5.450,148.985
C09841=1212.594,-46.106,-40.099,179.892,5.450,148.985
C09842=1212.600,-46.355,-40.087,179.890,5.450,148.986
C09843=1212.605,-46.605,-40.075,179.888,5.449,148.987
C09844=1212.610,-46.855,-40.062,179.885,5.449,148.988
C09845=1212.615,-47.105,-40.050,179.883,5.449,148.988
C09846=1212.620,-47.355,-40.038,179.880,5.449,148.989
C09847=1212.626,-47.604,-40.025,179.878,5.448,148.989
C09848=1212.631,-47.854,-40.013,179.876,5.448,148.990
C09849=1212.636,-48.103,-40.001,179.873,5.448,148.991
C09850=1212.642,-48.353,-39.989,179.871,5.448,148.992
C09851=1212.647,-48.623,-39.975,179.869,5.448,148.992
C09852=1212.652,-48.893,-39.963,179.865,5.448,148.993
C09853=1212.658,-49.163,-39.950,179.863,5.447,148.994
C09854=1212.663,-49.433,-39.935,179.860,5.447,148.995
C09855=1212.668,-49.683,-39.924,179.858,5.447,148.995
C09856=1212.673,-49.932,-39.912,179.855,5.447,148.996
C09857=1212.679,-50.182,-39.900,179.853,5.447,148.997
C09858=1212.684,-50.432,-39.888,179.851,5.446,148.997
C09859=1212.689,-50.681,-39.875,179.848,5.446,148.998
C09860=1212.695,-50.931,-39.863,179.846,5.446,148.999
C09861=1212.699,-51.180,-39.851,179.844,5.446,148.999
C09862=1212.705,-51.430,-39.839,179.841,5.445,149.000
C09863=1212.710,-51.679,-39.827,179.839,5.445,149.001
C09864=1212.715,-51.929,-39.815,179.836,5.445,149.001
C09865=1212.720,-52.179,-39.803,179.834,5.445,149.002
C09866=1212.726,-52.428,-39.790,179.832,5.445,149.003
C09867=1212.730,-52.678,-39.779,179.829,5.444,149.003
C09868=1212.735,-52.927,-39.767,179.827,5.445,149.004
C09869=1212.741,-53.177,-39.755,179.824,5.444,149.005
C09870=1212.746,-53.427,-39.743,179.822,5.443,149.005
C09871=1212.751,-53.676,-39.731,179.820,5.444,149.006
C09872=1212.756,-53.926,-39.719,179.817,5.443,149.007
C09873=1212.762,-54.176,-39.707,179.815,5.444,149.007
C09874=1212.767,-54.426,-39.694,179.812,5.443,149.008
C09875=1212.772,-54.675,-39.683,179.810,5.443,149.009
C09876=1212.777,-54.925,-39.671,179.808,5.443,149.010
C09877=1212.782,-55.174,-39.659,179.805,5.443,149.010
C09878=1212.787,-55.424,-39.647,179.802,5.442,149.011
C09879=1212.792,-55.674,-39.635,179.800,5.443,149.012
C09880=1212.797,-55.924,-39.624,179.798,5.442,149.012
C09881=1212.803,-56.173,-39.611,179.796,5.442,149.013
C09882=1212.808,-56.423,-39.599,179.793,5.442,149.014
C09883=1212.813,-56.673,-39.588,179.791,5.441,149.014
C09884=1212.818,-56.922,-39.575,179.789,5.441,149.015
C09885=1212.823,-57.172,-39.563,179.786,5.441,149.016
C09886=1212.828,-57.422,-39.552,179.784,5.441,149.016
C09887=1212.833,-57.672,-39.540,179.781,5.441,149.017
C09888=1212.839,-57.922,-39.528,179.779,5.440,149.018
C09889=1212.844,-58.171,-39.516,179.776,5.441,149.019
C09890=1212.849,-58.420,-39.504,179.774,5.440,149.019
C09891=1212.854,-58.670,-39.492,179.772,5.441,149.020
C09892=1212.859,-58.920,-39.481,179.770,5.440,149.020
C09893=1212.864,-59.169,-39.469,179.767,5.439,149.021
C09894=1212.869,-59.419,-39.457,179.765,5.440,149.022
C09895=1212.875,-59.669,-39.445,179.762,5.439,149.023
C09896=1212.879,-59.919,-39.434,179.760,5.440,149.023
C09897=1212.885,-60.168,-39.422,179.757,5.439,149.024
C09898=1212.890,-60.418,-39.411,179.755,5.439,149.025
C09899=1212.895,-60.667,-39.398,179.753,5.439,149.025
C09900=1212.901,-60.917,-39.386,179.750,5.439,149.026
C09901=1212.905,-61.167,-39.375,179.748,5.439,149.027
C09902=1212.911,-61.417,-39.363,179.746,5.438,149.027
C09903=1212.916,-61.666,-39.351,179.743,5.438,149.028
C09904=1212.921,-61.916,-39.340,179.741,5.438,149.029
C09905=1212.926,-62.166,-39.328,179.738,5.438,149.029
C09906=1212.931,-62.416,-39.317,179.736,5.438,149.030
C09907=1212.936,-62.666,-39.305,179.733,5.437,149.031
C09908=1212.942,-62.914,-39.293,179.731,5.437,149.031
C09909=1212.947,-63.164,-39.281,179.729,5.437,149.032
C09910=1212.952,-63.414,-39.269,179.726,5.437,149.033
C09911=1212.957,-63.663,-39.258,179.724,5.437,149.034
C09912=1212.962,-63.913,-39.246,179.722,5.436,149.034
C09913=1212.967,-64.163,-39.235,179.719,5.436,149.035
C09914=1212.973,-64.413,-39.223,179.717,5.436,149.035
C09915=1212.979,-64.662,-39.212,179.714,5.436,149.036
C09916=1212.983,-64.912,-39.200,179.712,5.436,149.037
C09917=1212.989,-65.162,-39.188,179.710,5.436,149.038
C09918=1212.993,-65.411,-39.177,179.707,5.435,149.038
C09919=1212.999,-65.661,-39.165,179.705,5.436,149.039
C09920=1213.004,-65.911,-39.154,179.702,5.435,149.040
C09921=1213.009,-66.161,-39.142,179.700,5.436,149.040
C09922=1213.014,-66.410,-39.131,179.698,5.435,149.041
C09923=1213.020,-66.660,-39.119,179.696,5.435,149.042
C09924=1213.024,-66.909,-39.108,179.693,5.435,149.042
C09925=1213.030,-67.159,-39.096,179.691,5.434,149.043
C09926=1213.035,-67.409,-39.085,179.688,5.435,149.044
C09927=1213.041,-67.658,-39.073,179.686,5.434,149.044
C09928=1213.045,-67.908,-39.062,179.684,5.434,149.045
C09929=1213.051,-68.158,-39.050,179.681,5.434,149.046
C09930=1213.055,-68.407,-39.039,179.678,5.434,149.047
C09931=1213.061,-68.657,-39.027,179.677,5.434,149.047
C09932=1213.066,-68.907,-39.017,179.674,5.433,149.048
C09933=1213.072,-69.157,-39.005,179.672,5.433,149.048
C09934=1213.076,-69.406,-38.993,179.669,5.433,149.049
C09935=1213.082,-69.656,-38.982,179.667,5.433,149.050
C09936=1213.087,-69.906,-38.970,179.665,5.433,149.051
C09937=1213.093,-70.155,-38.959,179.662,5.432,149.051
C09938=1213.097,-70.405,-38.947,179.660,5.433,149.052
C09939=1213.102,-70.654,-38.936,179.657,5.432,149.053
C09940=1213.108,-70.905,-38.925,179.656,5.432,149.053
C09941=1213.113,-71.154,-38.914,179.653,5.432,149.054
C09942=1213.118,-71.404,-38.902,179.651,5.432,149.055
C09943=1213.123,-71.653,-38.891,179.648,5.432,149.055
C09944=1213.129,-71.903,-38.879,179.645,5.431,149.056
C09945=1213.133,-72.153,-38.868,179.643,5.432,149.057
C09946=1213.139,-72.403,-38.858,179.641,5.431,149.057
C09947=1213.144,-72.652,-38.846,179.639,5.432,149.058
C09948=1213.149,-72.902,-38.834,179.636,5.431,149.059
C09949=1213.155,-73.151,-38.823,179.634,5.431,149.059
C09950=1213.160,-73.401,-38.812,179.632,5.431,149.060
C09951=1213.165,-73.651,-38.801,179.629,5.430,149.061
C09952=1213.170,-73.901,-38.789,179.627,5.431,149.061
C09953=1213.175,-74.150,-38.778,179.624,5.430,149.062
C09954=1213.180,-74.400,-38.767,179.622,5.431,149.063
C09955=1213.186,-74.671,-38.755,179.619,5.430,149.064
C09956=1213.192,-74.941,-38.743,179.617,5.430,149.064
C09957=1213.198,-75.212,-38.730,179.615,5.430,149.065
C09958=1213.203,-75.483,-38.718,179.612,5.430,149.066
C09959=1213.209,-75.732,-38.707,179.609,5.429,149.066
C09960=1213.213,-75.981,-38.696,179.607,5.429,149.067
C09961=1213.219,-76.231,-38.684,179.605,5.429,149.068
C09962=1213.224,-76.481,-38.674,179.603,5.429,149.068
C09963=1213.229,-76.731,-38.663,179.600,5.429,149.069
C09964=1213.234,-76.980,-38.651,179.598,5.429,149.070
C09965=1213.240,-77.230,-38.641,179.596,5.428,149.070
C09966=1213.245,-77.480,-38.629,179.594,5.429,149.071
C09967=1213.250,-77.730,-38.617,179.591,5.428,149.072
C09968=1213.256,-77.979,-38.607,179.588,5.428,149.073
C09969=1213.260,-78.229,-38.596,179.586,5.428,149.073
C09970=1213.265,-78.478,-38.585,179.583,5.428,149.074
C09971=1213.271,-78.729,-38.573,179.581,5.428,149.075
C09972=1213.276,-78.978,-38.562,179.579,5.428,149.075
C09973=1213.281,-79.227,-38.551,179.577,5.428,149.076
C09974=1213.286,-79.477,-38.541,179.574,5.427,149.077
C09975=1213.292,-79.727,-38.529,179.572,5.428,149.077
C09976=1213.297,-79.977,-38.519,179.570,5.427,149.078
C09977=1213.302,-80.226,-38.508,179.568,5.428,149.079
C09978=1213.307,-80.476,-38.496,179.565,5.427,149.079
C09979=1213.313,-80.726,-38.485,179.562,5.427,149.080
C09980=1213.318,-80.975,-38.474,179.560,5.427,149.081
C09981=1213.323,-81.225,-38.464,179.558,5.426,149.081
C09982=1213.327,-81.475,-38.452,179.556,5.427,149.082
C09983=1213.334,-81.725,-38.442,179.553,5.426,149.083
C09984=1213.339,-81.975,-38.430,179.551,5.427,149.083
C09985=1213.344,-82.224,-38.420,179.548,5.426,149.084
C09986=1213.349,-82.474,-38.409,179.546,5.426,149.085
C09987=1213.354,-82.723,-38.397,179.544,5.426,149.086
C09988=1213.360,-82.973,-38.387,179.542,5.426,149.086
C09989=1213.365,-83.223,-38.375,179.539,5.426,149.087
C09990=1213.370,-83.473,-38.365,179.537,5.425,149.087
C09991=1213.375,-83.722,-38.354,179.535,5.426,149.088
C09992=1213.380,-83.972,-38.343,179.532,5.425,149.089
C09993=1213.385,-84.221,-38.332,179.530,5.425,149.090
C09994=1213.390,-84.471,-38.322,179.527,5.425,149.090
C09995=1213.396,-84.722,-38.311,179.525,5.425,149.091
C09996=1213.401,-84.971,-38.300,179.523,5.425,149.091
//INST
///DATE 2021/06/15 17:23
///ATTR SC,RW,RJ
////FRAME ROBOT
///GROUP1 RB1
NOP
MOVL C00000 V=800.0 PL=0
MOVL C00001 V=800.0 PL=0
MOVL C00002 V=800.0 PL=0
MOVL C00003 V=800.0 PL=0
MOVL C00004 V=800.0 PL=0
MOVL C00005 V=800.0 PL=0
MOVL C00006 V=800.0 PL=0
MOVL C00007 V=800.0 PL=0
MOVL C00008 V=800.0 PL=0
MOVL C00009 V=800.0 PL=0
MOVL C00010 V=800.0 PL=0
MOVL C00011 V=800.0 PL=0
MOVL C00012 V=800.0 PL=0
MOVL C00013 V=800.0 PL=0
MOVL C00014 V=800.0 PL=0
MOVL C00015 V=800.0 PL=0
MOVL C00016 V=800.0 PL=0
MOVL C00017 V=800.0 PL=0
MOVL C00018 V=800.0 PL=0
MOVL C00019 V=800.0 PL=0
MOVL C00020 V=800.0 PL=0
MOVL C00021 V=800.0 PL=0
MOVL C00022 V=800.0 PL=0
MOVL C00023 V=800.0 PL=0
MOVL C00024 V=800.0 PL=0
MOVL C00025 V=800.0 PL=0
MOVL C00026 V=800.0 PL=0
MOVL C00027 V=800.0 PL=0
MOVL C00028 V=800.0 PL=0
MOVL C00029 V=800.0 PL=0
MOVL C00030 V=800.0 PL=0
MOVL C00031 V=800.0 PL=0
MOVL C00032 V=800.0 PL=0
MOVL C00033 V=800.0 PL=0
MOVL C00034 V=800.0 PL=0
MOVL C00035 V=800.0 PL=0
MOVL C00036 V=800.0 PL=0
MOVL C00037 V=800.0 PL=0
MOVL C00038 V=800.0 PL=0
MOVL C00039 V=800.0 PL=0
MOVL C00040 V=800.0 PL=0
MOVL C00041 V=800.0 PL=0
MOVL C00042 V=800.0 PL=0
MOVL C00043 V=800.0 PL=0
MOVL C00044 V=800.0 PL=0
MOVL C00045 V=800.0 PL=0
MOVL C00046 V=800.0 PL=0
MOVL C00047 V=800.0 PL=0
MOVL C00048 V=800.0 PL=0
MOVL C00049 V=800.0 PL=0
MOVL C00050 V=800.0 PL=0
MOVL C00051 V=800.0 PL=0
MOVL C00052 V=800.0 PL=0
MOVL C00053 V=800.0 PL=0
MOVL C00054 V=800.0 PL=0
MOVL C00055 V=800.0 PL=0
MOVL C00056 V=800.0 PL=0
MOVL C00057 V=800.0 PL=0
MOVL C00058 V=800.0 PL=0
MOVL C00059 V=800.0 PL=0
MOVL C00060 V=800.0 PL=0
MOVL C00061 V=800.0 PL=0
MOVL C00062 V=800.0 PL=0
MOVL C00063 V=800.0 PL=0
MOVL C00064 V=800.0 PL=0
MOVL C00065 V=800.0 PL=0
MOVL C00066 V=800.0 PL=0
MOVL C00067 V=800.0 PL=0
MOVL C00068 V=800.0 PL=0
MOVL C00069 V=800.0 PL=0
MOVL C00070 V=800.0 PL=0
MOVL C00071 V=800.0 PL=0
MOVL C00072 V=800.0 PL=0
MOVL C00073 V=800.0 PL=0
MOVL C00074 V=800.0 PL=0
MOVL C00075 V=800.0 PL=0
MOVL C00076 V=800.0 PL=0
MOVL C00077 V=800.0 PL=0
MOVL C00078 V=800.0 PL=0
MOVL C00079 V=800.0 PL=0
MOVL C00080 V=800.0 PL=0
MOVL C00081 V=800.0 PL=0
MOVL C00082 V=800.0 PL=0
MOVL C00083 V=800.0 PL=0
MOVL C00084 V=800.0 PL=0
MOVL C00085 V=800.0 PL=0
MOVL C00086 V=800.0 PL=0
MOVL C00087 V=800.0 PL=0
MOVL C00088 V=800.0 PL=0
MOVL C00089 V=800.0 PL=0
MOVL C00090 V=800.0 PL=0
MOVL C00091 V=800.0 PL=0
MOVL C00092 V=800.0 PL=0
MOVL C00093 V=800.0 PL=0
MOVL C00094 V=800.0 PL=0
MOVL C00095 V=800.0 PL=0
MOVL C00096 V=800.0 PL=0
MOVL C00097 V=800.0 PL=0
MOVL C00098 V=800.0 PL=0
MOVL C00099 V=800.0 PL=0
MOVL C00100 V=800.0 PL=0
MOVL C00101 V=800.0 PL=0
MOVL C00102 V=800.0 PL=0
MOVL C00103 V=800.0 PL=0
MOVL C00104 V=800.0 PL=0
MOVL C00105 V=800.0 PL=0
MOVL C00106 V=800.0 PL=0
MOVL C00107 V=800.0 PL=0
MOVL C00108 V=800.0 PL=0
MOVL C00109 V=800.0 PL=0
MOVL C00110 V=800.0 PL=0
MOVL C00111 V=800.0 PL=0
MOVL C00112 V=800.0 PL=0
MOVL C00113 V=800.0 PL=0
MOVL C00114 V=800.0 PL=0
MOVL C00115 V=800.0 PL=0
MOVL C00116 V=800.0 PL=0
MOVL C00117 V=800.0 PL=0
MOVL C00118 V=800.0 PL=0
MOVL C00119 V=800.0 PL=0
MOVL C00120 V=800.0 PL=0
MOVL C00121 V=800.0 PL=0
MOVL C00122 V=800.0 PL=0
MOVL C00123 V=800.0 PL=0
MOVL C00124 V=800.0 PL=0
MOVL C00125 V=800.0 PL=0
MOVL C00126 V=800.0 PL=0
MOVL C00127 V=800.0 PL=0
MOVL C00128 V=800.0 PL=0
MOVL C00129 V=800.0 PL=0
MOVL C00130 V=800.0 PL=0
MOVL C00131 V=800.0 PL=0
MOVL C00132 V=800.0 PL=0
MOVL C00133 V=800.0 PL=0
MOVL C00134 V=800.0 PL=0
MOVL C00135 V=800.0 PL=0
MOVL C00136 V=800.0 PL=0
MOVL C00137 V=800.0 PL=0
MOVL C00138 V=800.0 PL=0
MOVL C00139 V=800.0 PL=0
MOVL C00140 V=800.0 PL=0
MOVL C00141 V=800.0 PL=0
MOVL C00142 V=800.0 PL=0
MOVL C00143 V=800.0 PL=0
MOVL C00144 V=800.0 PL=0
MOVL C00145 V=800.0 PL=0
MOVL C00146 V=800.0 PL=0
MOVL C00147 V=800.0 PL=0
MOVL C00148 V=800.0 PL=0
MOVL C00149 V=800.0 PL=0
MOVL C00150 V=800.0 PL=0
MOVL C00151 V=800.0 PL=0
MOVL C00152 V=800.0 PL=0
MOVL C00153 V=800.0 PL=0
MOVL C00154 V=800.0 PL=0
MOVL C00155 V=800.0 PL=0
MOVL C00156 V=800.0 PL=0
MOVL C00157 V=800.0 PL=0
MOVL C00158 V=800.0 PL=0
MOVL C00159 V=800.0 PL=0
MOVL C00160 V=800.0 PL=0
MOVL C00161 V=800.0 PL=0
MOVL C00162 V=800.0 PL=0
MOVL C00163 V=800.0 PL=0
MOVL C00164 V=800.0 PL=0
MOVL C00165 V=800.0 PL=0
MOVL C00166 V=800.0 PL=0
MOVL C00167 V=800.0 PL=0
MOVL C00168 V=800.0 PL=0
MOVL C00169 V=800.0 PL=0
MOVL C00170 V=800.0 PL=0
MOVL C00171 V=800.0 PL=0
MOVL C00172 V=800.0 PL=0
MOVL C00173 V=800.0 PL=0
MOVL C00174 V=800.0 PL=0
MOVL C00175 V=800.0 PL=0
MOVL C00176 V=800.0 PL=0
MOVL C00177 V=800.0 PL=0
MOVL C00178 V=800.0 PL=0
MOVL C00179 V=800.0 PL=0
MOVL C00180 V=800.0 PL=0
MOVL C00181 V=800.0 PL=0
MOVL C00182 V=800.0 PL=0
MOVL C00183 V=800.0 PL=0
MOVL C00184 V=800.0 PL=0
MOVL C00185 V=800.0 PL=0
MOVL C00186 V=800.0 PL=0
MOVL C00187 V=800.0 PL=0
MOVL C00188 V=800.0 PL=0
MOVL C00189 V=800.0 PL=0
MOVL C00190 V=800.0 PL=0
MOVL C00191 V=800.0 PL=0
MOVL C00192 V=800.0 PL=0
MOVL C00193 V=800.0 PL=0
MOVL C00194 V=800.0 PL=0
MOVL C00195 V=800.0 PL=0
MOVL C00196 V=800.0 PL=0
MOVL C00197 V=800.0 PL=0
MOVL C00198 V=800.0 PL=0
MOVL C00199 V=800.0 PL=0
MOVL C00200 V=800.0 PL=0
MOVL C00201 V=800.0 PL=0
MOVL C00202 V=800.0 PL=0
MOVL C00203 V=800.0 PL=0
MOVL C00204 V=800.0 PL=0
MOVL C00205 V=800.0 PL=0
MOVL C00206 V=800.0 PL=0
MOVL C00207 V=800.0 PL=0
MOVL C00208 V=800.0 PL=0
MOVL C00209 V=800.0 PL=0
MOVL C00210 V=800.0 PL=0
MOVL C00211 V=800.0 PL=0
MOVL C00212 V=800.0 PL=0
MOVL C00213 V=800.0 PL=0
MOVL C00214 V=800.0 PL=0
MOVL C00215 V=800.0 PL=0
MOVL C00216 V=800.0 PL=0
MOVL C00217 V=800.0 PL=0
MOVL C00218 V=800.0 PL=0
MOVL C00219 V=800.0 PL=0
MOVL C00220 V=800.0 PL=0
MOVL C00221 V=800.0 PL=0
MOVL C00222 V=800.0 PL=0
MOVL C00223 V=800.0 PL=0
MOVL C00224 V=800.0 PL=0
MOVL C00225 V=800.0 PL=0
MOVL C00226 V=800.0 PL=0
MOVL C00227 V=800.0 PL=0
MOVL C00228 V=800.0 PL=0
MOVL C00229 V=800.0 PL=0
MOVL C00230 V=800.0 PL=0
MOVL C00231 V=800.0 PL=0
MOVL C00232 V=800.0 PL=0
MOVL C00233 V=800.0 PL=0
MOVL C00234 V=800.0 PL=0
MOVL C00235 V=800.0 PL=0
MOVL C00236 V=800.0 PL=0
MOVL C00237 V=800.0 PL=0
MOVL C00238 V=800.0 PL=0
MOVL C00239 V=800.0 PL=0
MOVL C00240 V=800.0 PL=0
MOVL C00241 V=800.0 PL=0
MOVL C00242 V=800.0 PL=0
MOVL C00243 V=800.0 PL=0
MOVL C00244 V=800.0 PL=0
MOVL C00245 V=800.0 PL=0
MOVL C00246 V=800.0 PL=0
MOVL C00247 V=800.0 PL=0
MOVL C00248 V=800.0 PL=0
MOVL C00249 V=800.0 PL=0
MOVL C00250 V=800.0 PL=0
MOVL C00251 V=800.0 PL=0
MOVL C00252 V=800.0 PL=0
MOVL C00253 V=800.0 PL=0
MOVL C00254 V=800.0 PL=0
MOVL C00255 V=800.0 PL=0
MOVL C00256 V=800.0 PL=0
MOVL C00257 V=800.0 PL=0
MOVL C00258 V=800.0 PL=0
MOVL C00259 V=800.0 PL=0
MOVL C00260 V=800.0 PL=0
MOVL C00261 V=800.0 PL=0
MOVL C00262 V=800.0 PL=0
MOVL C00263 V=800.0 PL=0
MOVL C00264 V=800.0 PL=0
MOVL C00265 V=800.0 PL=0
MOVL C00266 V=800.0 PL=0
MOVL C00267 V=800.0 PL=0
MOVL C00268 V=800.0 PL=0
MOVL C00269 V=800.0 PL=0
MOVL C00270 V=800.0 PL=0
MOVL C00271 V=800.0 PL=0
MOVL C00272 V=800.0 PL=0
MOVL C00273 V=800.0 PL=0
MOVL C00274 V=800.0 PL=0
MOVL C00275 V=800.0 PL=0
MOVL C00276 V=800.0 PL=0
MOVL C00277 V=800.0 PL=0
MOVL C00278 V=800.0 PL=0
MOVL C00279 V=800.0 PL=0
MOVL C00280 V=800.0 PL=0
MOVL C00281 V=800.0 PL=0
MOVL C00282 V=800.0 PL=0
MOVL C00283 V=800.0 PL=0
MOVL C00284 V=800.0 PL=0
MOVL C00285 V=800.0 PL=0
MOVL C00286 V=800.0 PL=0
MOVL C00287 V=800.0 PL=0
MOVL C00288 V=800.0 PL=0
MOVL C00289 V=800.0 PL=0
MOVL C00290 V=800.0 PL=0
MOVL C00291 V=800.0 PL=0
MOVL C00292 V=800.0 PL=0
MOVL C00293 V=800.0 PL=0
MOVL C00294 V=800.0 PL=0
MOVL C00295 V=800.0 PL=0
MOVL C00296 V=800.0 PL=0
MOVL C00297 V=800.0 PL=0
MOVL C00298 V=800.0 PL=0
MOVL C00299 V=800.0 PL=0
MOVL C00300 V=800.0 PL=0
MOVL C00301 V=800.0 PL=0
MOVL C00302 V=800.0 PL=0
MOVL C00303 V=800.0 PL=0
MOVL C00304 V=800.0 PL=0
MOVL C00305 V=800.0 PL=0
MOVL C00306 V=800.0 PL=0
MOVL C00307 V=800.0 PL=0
MOVL C00308 V=800.0 PL=0
MOVL C00309 V=800.0 PL=0
MOVL C00310 V=800.0 PL=0
MOVL C00311 V=800.0 PL=0
MOVL C00312 V=800.0 PL=0
MOVL C00313 V=800.0 PL=0
MOVL C00314 V=800.0 PL=0
MOVL C00315 V=800.0 PL=0
MOVL C00316 V=800.0 PL=0
MOVL C00317 V=800.0 PL=0
MOVL C00318 V=800.0 PL=0
MOVL C00319 V=800.0 PL=0
MOVL C00320 V=800.0 PL=0
MOVL C00321 V=800.0 PL=0
MOVL C00322 V=800.0 PL=0
MOVL C00323 V=800.0 PL=0
MOVL C00324 V=800.0 PL=0
MOVL C00325 V=800.0 PL=0
MOVL C00326 V=800.0 PL=0
MOVL C00327 V=800.0 PL=0
MOVL C00328 V=800.0 PL=0
MOVL C00329 V=800.0 PL=0
MOVL C00330 V=800.0 PL=0
MOVL C00331 V=800.0 PL=0
MOVL C00332 V=800.0 PL=0
MOVL C00333 V=800.0 PL=0
MOVL C00334 V=800.0 PL=0
MOVL C00335 V=800.0 PL=0
MOVL C00336 V=800.0 PL=0
MOVL C00337 V=800.0 PL=0
MOVL C00338 V=800.0 PL=0
MOVL C00339 V=800.0 PL=0
MOVL C00340 V=800.0 PL=0
MOVL C00341 V=800.0 PL=0
MOVL C00342 V=800.0 PL=0
MOVL C00343 V=800.0 PL=0
MOVL C00344 V=800.0 PL=0
MOVL C00345 V=800.0 PL=0
MOVL C00346 V=800.0 PL=0
MOVL C00347 V=800.0 PL=0
MOVL C00348 V=800.0 PL=0
MOVL C00349 V=800.0 PL=0
MOVL C00350 V=800.0 PL=0
MOVL C00351 V=800.0 PL=0
MOVL C00352 V=800.0 PL=0
MOVL C00353 V=800.0 PL=0
MOVL C00354 V=800.0 PL=0
MOVL C00355 V=800.0 PL=0
MOVL C00356 V=800.0 PL=0
MOVL C00357 V=800.0 PL=0
MOVL C00358 V=800.0 PL=0
MOVL C00359 V=800.0 PL=0
MOVL C00360 V=800.0 PL=0
MOVL C00361 V=800.0 PL=0
MOVL C00362 V=800.0 PL=0
MOVL C00363 V=800.0 PL=0
MOVL C00364 V=800.0 PL=0
MOVL C00365 V=800.0 PL=0
MOVL C00366 V=800.0 PL=0
MOVL C00367 V=800.0 PL=0
MOVL C00368 V=800.0 PL=0
MOVL C00369 V=800.0 PL=0
MOVL C00370 V=800.0 PL=0
MOVL C00371 V=800.0 PL=0
MOVL C00372 V=800.0 PL=0
MOVL C00373 V=800.0 PL=0
MOVL C00374 V=800.0 PL=0
MOVL C00375 V=800.0 PL=0
MOVL C00376 V=800.0 PL=0
MOVL C00377 V=800.0 PL=0
MOVL C00378 V=800.0 PL=0
MOVL C00379 V=800.0 PL=0
MOVL C00380 V=800.0 PL=0
MOVL C00381 V=800.0 PL=0
MOVL C00382 V=800.0 PL=0
MOVL C00383 V=800.0 PL=0
MOVL C00384 V=800.0 PL=0
MOVL C00385 V=800.0 PL=0
MOVL C00386 V=800.0 PL=0
MOVL C00387 V=800.0 PL=0
MOVL C00388 V=800.0 PL=0
MOVL C00389 V=800.0 PL=0
MOVL C00390 V=800.0 PL=0
MOVL C00391 V=800.0 PL=0
MOVL C00392 V=800.0 PL=0
MOVL C00393 V=800.0 PL=0
MOVL C00394 V=800.0 PL=0
MOVL C00395 V=800.0 PL=0
MOVL C00396 V=800.0 PL=0
MOVL C00397 V=800.0 PL=0
MOVL C00398 V=800.0 PL=0
MOVL C00399 V=800.0 PL=0
MOVL C00400 V=800.0 PL=0
MOVL C00401 V=800.0 PL=0
MOVL C00402 V=800.0 PL=0
MOVL C00403 V=800.0 PL=0
MOVL C00404 V=800.0 PL=0
MOVL C00405 V=800.0 PL=0
MOVL C00406 V=800.0 PL=0
MOVL C00407 V=800.0 PL=0
MOVL C00408 V=800.0 PL=0
MOVL C00409 V=800.0 PL=0
MOVL C00410 V=800.0 PL=0
MOVL C00411 V=800.0 PL=0
MOVL C00412 V=800.0 PL=0
MOVL C00413 V=800.0 PL=0
MOVL C00414 V=800.0 PL=0
MOVL C00415 V=800.0 PL=0
MOVL C00416 V=800.0 PL=0
MOVL C00417 V=800.0 PL=0
MOVL C00418 V=800.0 PL=0
MOVL C00419 V=800.0 PL=0
MOVL C00420 V=800.0 PL=0
MOVL C00421 V=800.0 PL=0
MOVL C00422 V=800.0 PL=0
MOVL C00423 V=800.0 PL=0
MOVL C00424 V=800.0 PL=0
MOVL C00425 V=800.0 PL=0
MOVL C00426 V=800.0 PL=0
MOVL C00427 V=800.0 PL=0
MOVL C00428 V=800.0 PL=0
MOVL C00429 V=800.0 PL=0
MOVL C00430 V=800.0 PL=0
MOVL C00431 V=800.0 PL=0
MOVL C00432 V=800.0 PL=0
MOVL C00433 V=800.0 PL=0
MOVL C00434 V=800.0 PL=0
MOVL C00435 V=800.0 PL=0
MOVL C00436 V=800.0 PL=0
MOVL C00437 V=800.0 PL=0
MOVL C00438 V=800.0 PL=0
MOVL C00439 V=800.0 PL=0
MOVL C00440 V=800.0 PL=0
MOVL C00441 V=800.0 PL=0
MOVL C00442 V=800.0 PL=0
MOVL C00443 V=800.0 PL=0
MOVL C00444 V=800.0 PL=0
MOVL C00445 V=800.0 PL=0
MOVL C00446 V=800.0 PL=0
MOVL C00447 V=800.0 PL=0
MOVL C00448 V=800.0 PL=0
MOVL C00449 V=800.0 PL=0
MOVL C00450 V=800.0 PL=0
MOVL C00451 V=800.0 PL=0
MOVL C00452 V=800.0 PL=0
MOVL C00453 V=800.0 PL=0
MOVL C00454 V=800.0 PL=0
MOVL C00455 V=800.0 PL=0
MOVL C00456 V=800.0 PL=0
MOVL C00457 V=800.0 PL=0
MOVL C00458 V=800.0 PL=0
MOVL C00459 V=800.0 PL=0
MOVL C00460 V=800.0 PL=0
MOVL C00461 V=800.0 PL=0
MOVL C00462 V=800.0 PL=0
MOVL C00463 V=800.0 PL=0
MOVL C00464 V=800.0 PL=0
MOVL C00465 V=800.0 PL=0
MOVL C00466 V=800.0 PL=0
MOVL C00467 V=800.0 PL=0
MOVL C00468 V=800.0 PL=0
MOVL C00469 V=800.0 PL=0
MOVL C00470 V=800.0 PL=0
MOVL C00471 V=800.0 PL=0
MOVL C00472 V=800.0 PL=0
MOVL C00473 V=800.0 PL=0
MOVL C00474 V=800.0 PL=0
MOVL C00475 V=800.0 PL=0
MOVL C00476 V=800.0 PL=0
MOVL C00477 V=800.0 PL=0
MOVL C00478 V=800.0 PL=0
MOVL C00479 V=800.0 PL=0
MOVL C00480 V=800.0 PL=0
MOVL C00481 V=800.0 PL=0
MOVL C00482 V=800.0 PL=0
MOVL C00483 V=800.0 PL=0
MOVL C00484 V=800.0 PL=0
MOVL C00485 V=800.0 PL=0
MOVL C00486 V=800.0 PL=0
MOVL C00487 V=800.0 PL=0
MOVL C00488 V=800.0 PL=0
MOVL C00489 V=800.0 PL=0
MOVL C00490 V=800.0 PL=0
MOVL C00491 V=800.0 PL=0
MOVL C00492 V=800.0 PL=0
MOVL C00493 V=800.0 PL=0
MOVL C00494 V=800.0 PL=0
MOVL C00495 V=800.0 PL=0
MOVL C00496 V=800.0 PL=0
MOVL C00497 V=800.0 PL=0
MOVL C00498 V=800.0 PL=0
MOVL C00499 V=800.0 PL=0
MOVL C00500 V=800.0 PL=0
MOVL C00501 V=800.0 PL=0
MOVL C00502 V=800.0 PL=0
MOVL C00503 V=800.0 PL=0
MOVL C00504 V=800.0 PL=0
MOVL C00505 V=800.0 PL=0
MOVL C00506 V=800.0 PL=0
MOVL C00507 V=800.0 PL=0
MOVL C00508 V=800.0 PL=0
MOVL C00509 V=800.0 PL=0
MOVL C00510 V=800.0 PL=0
MOVL C00511 V=800.0 PL=0
MOVL C00512 V=800.0 PL=0
MOVL C00513 V=800.0 PL=0
MOVL C00514 V=800.0 PL=0
MOVL C00515 V=800.0 PL=0
MOVL C00516 V=800.0 PL=0
MOVL C00517 V=800.0 PL=0
MOVL C00518 V=800.0 PL=0
MOVL C00519 V=800.0 PL=0
MOVL C00520 V=800.0 PL=0
MOVL C00521 V=800.0 PL=0
MOVL C00522 V=800.0 PL=0
MOVL C00523 V=800.0 PL=0
MOVL C00524 V=800.0 PL=0
MOVL C00525 V=800.0 PL=0
MOVL C00526 V=800.0 PL=0
MOVL C00527 V=800.0 PL=0
MOVL C00528 V=800.0 PL=0
MOVL C00529 V=800.0 PL=0
MOVL C00530 V=800.0 PL=0
MOVL C00531 V=800.0 PL=0
MOVL C00532 V=800.0 PL=0
MOVL C00533 V=800.0 PL=0
MOVL C00534 V=800.0 PL=0
MOVL C00535 V=800.0 PL=0
MOVL C00536 V=800.0 PL=0
MOVL C00537 V=800.0 PL=0
MOVL C00538 V=800.0 PL=0
MOVL C00539 V=800.0 PL=0
MOVL C00540 V=800.0 PL=0
MOVL C00541 V=800.0 PL=0
MOVL C00542 V=800.0 PL=0
MOVL C00543 V=800.0 PL=0
MOVL C00544 V=800.0 PL=0
MOVL C00545 V=800.0 PL=0
MOVL C00546 V=800.0 PL=0
MOVL C00547 V=800.0 PL=0
MOVL C00548 V=800.0 PL=0
MOVL C00549 V=800.0 PL=0
MOVL C00550 V=800.0 PL=0
MOVL C00551 V=800.0 PL=0
MOVL C00552 V=800.0 PL=0
MOVL C00553 V=800.0 PL=0
MOVL C00554 V=800.0 PL=0
MOVL C00555 V=800.0 PL=0
MOVL C00556 V=800.0 PL=0
MOVL C00557 V=800.0 PL=0
MOVL C00558 V=800.0 PL=0
MOVL C00559 V=800.0 PL=0
MOVL C00560 V=800.0 PL=0
MOVL C00561 V=800.0 PL=0
MOVL C00562 V=800.0 PL=0
MOVL C00563 V=800.0 PL=0
MOVL C00564 V=800.0 PL=0
MOVL C00565 V=800.0 PL=0
MOVL C00566 V=800.0 PL=0
MOVL C00567 V=800.0 PL=0
MOVL C00568 V=800.0 PL=0
MOVL C00569 V=800.0 PL=0
MOVL C00570 V=800.0 PL=0
MOVL C00571 V=800.0 PL=0
MOVL C00572 V=800.0 PL=0
MOVL C00573 V=800.0 PL=0
MOVL C00574 V=800.0 PL=0
MOVL C00575 V=800.0 PL=0
MOVL C00576 V=800.0 PL=0
MOVL C00577 V=800.0 PL=0
MOVL C00578 V=800.0 PL=0
MOVL C00579 V=800.0 PL=0
MOVL C00580 V=800.0 PL=0
MOVL C00581 V=800.0 PL=0
MOVL C00582 V=800.0 PL=0
MOVL C00583 V=800.0 PL=0
MOVL C00584 V=800.0 PL=0
MOVL C00585 V=800.0 PL=0
MOVL C00586 V=800.0 PL=0
MOVL C00587 V=800.0 PL=0
MOVL C00588 V=800.0 PL=0
MOVL C00589 V=800.0 PL=0
MOVL C00590 V=800.0 PL=0
MOVL C00591 V=800.0 PL=0
MOVL C00592 V=800.0 PL=0
MOVL C00593 V=800.0 PL=0
MOVL C00594 V=800.0 PL=0
MOVL C00595 V=800.0 PL=0
MOVL C00596 V=800.0 PL=0
MOVL C00597 V=800.0 PL=0
MOVL C00598 V=800.0 PL=0
MOVL C00599 V=800.0 PL=0
MOVL C00600 V=800.0 PL=0
MOVL C00601 V=800.0 PL=0
MOVL C00602 V=800.0 PL=0
MOVL C00603 V=800.0 PL=0
MOVL C00604 V=800.0 PL=0
MOVL C00605 V=800.0 PL=0
MOVL C00606 V=800.0 PL=0
MOVL C00607 V=800.0 PL=0
MOVL C00608 V=800.0 PL=0
MOVL C00609 V=800.0 PL=0
MOVL C00610 V=800.0 PL=0
MOVL C00611 V=800.0 PL=0
MOVL C00612 V=800.0 PL=0
MOVL C00613 V=800.0 PL=0
MOVL C00614 V=800.0 PL=0
MOVL C00615 V=800.0 PL=0
MOVL C00616 V=800.0 PL=0
MOVL C00617 V=800.0 PL=0
MOVL C00618 V=800.0 PL=0
MOVL C00619 V=800.0 PL=0
MOVL C00620 V=800.0 PL=0
MOVL C00621 V=800.0 PL=0
MOVL C00622 V=800.0 PL=0
MOVL C00623 V=800.0 PL=0
MOVL C00624 V=800.0 PL=0
MOVL C00625 V=800.0 PL=0
MOVL C00626 V=800.0 PL=0
MOVL C00627 V=800.0 PL=0
MOVL C00628 V=800.0 PL=0
MOVL C00629 V=800.0 PL=0
MOVL C00630 V=800.0 PL=0
MOVL C00631 V=800.0 PL=0
MOVL C00632 V=800.0 PL=0
MOVL C00633 V=800.0 PL=0
MOVL C00634 V=800.0 PL=0
MOVL C00635 V=800.0 PL=0
MOVL C00636 V=800.0 PL=0
MOVL C00637 V=800.0 PL=0
MOVL C00638 V=800.0 PL=0
MOVL C00639 V=800.0 PL=0
MOVL C00640 V=800.0 PL=0
MOVL C00641 V=800.0 PL=0
MOVL C00642 V=800.0 PL=0
MOVL C00643 V=800.0 PL=0
MOVL C00644 V=800.0 PL=0
MOVL C00645 V=800.0 PL=0
MOVL C00646 V=800.0 PL=0
MOVL C00647 V=800.0 PL=0
MOVL C00648 V=800.0 PL=0
MOVL C00649 V=800.0 PL=0
MOVL C00650 V=800.0 PL=0
MOVL C00651 V=800.0 PL=0
MOVL C00652 V=800.0 PL=0
MOVL C00653 V=800.0 PL=0
MOVL C00654 V=800.0 PL=0
MOVL C00655 V=800.0 PL=0
MOVL C00656 V=800.0 PL=0
MOVL C00657 V=800.0 PL=0
MOVL C00658 V=800.0 PL=0
MOVL C00659 V=800.0 PL=0
MOVL C00660 V=800.0 PL=0
MOVL C00661 V=800.0 PL=0
MOVL C00662 V=800.0 PL=0
MOVL C00663 V=800.0 PL=0
MOVL C00664 V=800.0 PL=0
MOVL C00665 V=800.0 PL=0
MOVL C00666 V=800.0 PL=0
MOVL C00667 V=800.0 PL=0
MOVL C00668 V=800.0 PL=0
MOVL C00669 V=800.0 PL=0
MOVL C00670 V=800.0 PL=0
MOVL C00671 V=800.0 PL=0
MOVL C00672 V=800.0 PL=0
MOVL C00673 V=800.0 PL=0
MOVL C00674 V=800.0 PL=0
MOVL C00675 V=800.0 PL=0
MOVL C00676 V=800.0 PL=0
MOVL C00677 V=800.0 PL=0
MOVL C00678 V=800.0 PL=0
MOVL C00679 V=800.0 PL=0
MOVL C00680 V=800.0 PL=0
MOVL C00681 V=800.0 PL=0
MOVL C00682 V=800.0 PL=0
MOVL C00683 V=800.0 PL=0
MOVL C00684 V=800.0 PL=0
MOVL C00685 V=800.0 PL=0
MOVL C00686 V=800.0 PL=0
MOVL C00687 V=800.0 PL=0
MOVL C00688 V=800.0 PL=0
MOVL C00689 V=800.0 PL=0
MOVL C00690 V=800.0 PL=0
MOVL C00691 V=800.0 PL=0
MOVL C00692 V=800.0 PL=0
MOVL C00693 V=800.0 PL=0
MOVL C00694 V=800.0 PL=0
MOVL C00695 V=800.0 PL=0
MOVL C00696 V=800.0 PL=0
MOVL C00697 V=800.0 PL=0
MOVL C00698 V=800.0 PL=0
MOVL C00699 V=800.0 PL=0
MOVL C00700 V=800.0 PL=0
MOVL C00701 V=800.0 PL=0
MOVL C00702 V=800.0 PL=0
MOVL C00703 V=800.0 PL=0
MOVL C00704 V=800.0 PL=0
MOVL C00705 V=800.0 PL=0
MOVL C00706 V=800.0 PL=0
MOVL C00707 V=800.0 PL=0
MOVL C00708 V=800.0 PL=0
MOVL C00709 V=800.0 PL=0
MOVL C00710 V=800.0 PL=0
MOVL C00711 V=800.0 PL=0
MOVL C00712 V=800.0 PL=0
MOVL C00713 V=800.0 PL=0
MOVL C00714 V=800.0 PL=0
MOVL C00715 V=800.0 PL=0
MOVL C00716 V=800.0 PL=0
MOVL C00717 V=800.0 PL=0
MOVL C00718 V=800.0 PL=0
MOVL C00719 V=800.0 PL=0
MOVL C00720 V=800.0 PL=0
MOVL C00721 V=800.0 PL=0
MOVL C00722 V=800.0 PL=0
MOVL C00723 V=800.0 PL=0
MOVL C00724 V=800.0 PL=0
MOVL C00725 V=800.0 PL=0
MOVL C00726 V=800.0 PL=0
MOVL C00727 V=800.0 PL=0
MOVL C00728 V=800.0 PL=0
MOVL C00729 V=800.0 PL=0
MOVL C00730 V=800.0 PL=0
MOVL C00731 V=800.0 PL=0
MOVL C00732 V=800.0 PL=0
MOVL C00733 V=800.0 PL=0
MOVL C00734 V=800.0 PL=0
MOVL C00735 V=800.0 PL=0
MOVL C00736 V=800.0 PL=0
MOVL C00737 V=800.0 PL=0
MOVL C00738 V=800.0 PL=0
MOVL C00739 V=800.0 PL=0
MOVL C00740 V=800.0 PL=0
MOVL C00741 V=800.0 PL=0
MOVL C00742 V=800.0 PL=0
MOVL C00743 V=800.0 PL=0
MOVL C00744 V=800.0 PL=0
MOVL C00745 V=800.0 PL=0
MOVL C00746 V=800.0 PL=0
MOVL C00747 V=800.0 PL=0
MOVL C00748 V=800.0 PL=0
MOVL C00749 V=800.0 PL=0
MOVL C00750 V=800.0 PL=0
MOVL C00751 V=800.0 PL=0
MOVL C00752 V=800.0 PL=0
MOVL C00753 V=800.0 PL=0
MOVL C00754 V=800.0 PL=0
MOVL C00755 V=800.0 PL=0
MOVL C00756 V=800.0 PL=0
MOVL C00757 V=800.0 PL=0
MOVL C00758 V=800.0 PL=0
MOVL C00759 V=800.0 PL=0
MOVL C00760 V=800.0 PL=0
MOVL C00761 V=800.0 PL=0
MOVL C00762 V=800.0 PL=0
MOVL C00763 V=800.0 PL=0
MOVL C00764 V=800.0 PL=0
MOVL C00765 V=800.0 PL=0
MOVL C00766 V=800.0 PL=0
MOVL C00767 V=800.0 PL=0
MOVL C00768 V=800.0 PL=0
MOVL C00769 V=800.0 PL=0
MOVL C00770 V=800.0 PL=0
MOVL C00771 V=800.0 PL=0
MOVL C00772 V=800.0 PL=0
MOVL C00773 V=800.0 PL=0
MOVL C00774 V=800.0 PL=0
MOVL C00775 V=800.0 PL=0
MOVL C00776 V=800.0 PL=0
MOVL C00777 V=800.0 PL=0
MOVL C00778 V=800.0 PL=0
MOVL C00779 V=800.0 PL=0
MOVL C00780 V=800.0 PL=0
MOVL C00781 V=800.0 PL=0
MOVL C00782 V=800.0 PL=0
MOVL C00783 V=800.0 PL=0
MOVL C00784 V=800.0 PL=0
MOVL C00785 V=800.0 PL=0
MOVL C00786 V=800.0 PL=0
MOVL C00787 V=800.0 PL=0
MOVL C00788 V=800.0 PL=0
MOVL C00789 V=800.0 PL=0
MOVL C00790 V=800.0 PL=0
MOVL C00791 V=800.0 PL=0
MOVL C00792 V=800.0 PL=0
MOVL C00793 V=800.0 PL=0
MOVL C00794 V=800.0 PL=0
MOVL C00795 V=800.0 PL=0
MOVL C00796 V=800.0 PL=0
MOVL C00797 V=800.0 PL=0
MOVL C00798 V=800.0 PL=0
MOVL C00799 V=800.0 PL=0
MOVL C00800 V=800.0 PL=0
MOVL C00801 V=800.0 PL=0
MOVL C00802 V=800.0 PL=0
MOVL C00803 V=800.0 PL=0
MOVL C00804 V=800.0 PL=0
MOVL C00805 V=800.0 PL=0
MOVL C00806 V=800.0 PL=0
MOVL C00807 V=800.0 PL=0
MOVL C00808 V=800.0 PL=0
MOVL C00809 V=800.0 PL=0
MOVL C00810 V=800.0 PL=0
MOVL C00811 V=800.0 PL=0
MOVL C00812 V=800.0 PL=0
MOVL C00813 V=800.0 PL=0
MOVL C00814 V=800.0 PL=0
MOVL C00815 V=800.0 PL=0
MOVL C00816 V=800.0 PL=0
MOVL C00817 V=800.0 PL=0
MOVL C00818 V=800.0 PL=0
MOVL C00819 V=800.0 PL=0
MOVL C00820 V=800.0 PL=0
MOVL C00821 V=800.0 PL=0
MOVL C00822 V=800.0 PL=0
MOVL C00823 V=800.0 PL=0
MOVL C00824 V=800.0 PL=0
MOVL C00825 V=800.0 PL=0
MOVL C00826 V=800.0 PL=0
MOVL C00827 V=800.0 PL=0
MOVL C00828 V=800.0 PL=0
MOVL C00829 V=800.0 PL=0
MOVL C00830 V=800.0 PL=0
MOVL C00831 V=800.0 PL=0
MOVL C00832 V=800.0 PL=0
MOVL C00833 V=800.0 PL=0
MOVL C00834 V=800.0 PL=0
MOVL C00835 V=800.0 PL=0
MOVL C00836 V=800.0 PL=0
MOVL C00837 V=800.0 PL=0
MOVL C00838 V=800.0 PL=0
MOVL C00839 V=800.0 PL=0
MOVL C00840 V=800.0 PL=0
MOVL C00841 V=800.0 PL=0
MOVL C00842 V=800.0 PL=0
MOVL C00843 V=800.0 PL=0
MOVL C00844 V=800.0 PL=0
MOVL C00845 V=800.0 PL=0
MOVL C00846 V=800.0 PL=0
MOVL C00847 V=800.0 PL=0
MOVL C00848 V=800.0 PL=0
MOVL C00849 V=800.0 PL=0
MOVL C00850 V=800.0 PL=0
MOVL C00851 V=800.0 PL=0
MOVL C00852 V=800.0 PL=0
MOVL C00853 V=800.0 PL=0
MOVL C00854 V=800.0 PL=0
MOVL C00855 V=800.0 PL=0
MOVL C00856 V=800.0 PL=0
MOVL C00857 V=800.0 PL=0
MOVL C00858 V=800.0 PL=0
MOVL C00859 V=800.0 PL=0
MOVL C00860 V=800.0 PL=0
MOVL C00861 V=800.0 PL=0
MOVL C00862 V=800.0 PL=0
MOVL C00863 V=800.0 PL=0
MOVL C00864 V=800.0 PL=0
MOVL C00865 V=800.0 PL=0
MOVL C00866 V=800.0 PL=0
MOVL C00867 V=800.0 PL=0
MOVL C00868 V=800.0 PL=0
MOVL C00869 V=800.0 PL=0
MOVL C00870 V=800.0 PL=0
MOVL C00871 V=800.0 PL=0
MOVL C00872 V=800.0 PL=0
MOVL C00873 V=800.0 PL=0
MOVL C00874 V=800.0 PL=0
MOVL C00875 V=800.0 PL=0
MOVL C00876 V=800.0 PL=0
MOVL C00877 V=800.0 PL=0
MOVL C00878 V=800.0 PL=0
MOVL C00879 V=800.0 PL=0
MOVL C00880 V=800.0 PL=0
MOVL C00881 V=800.0 PL=0
MOVL C00882 V=800.0 PL=0
MOVL C00883 V=800.0 PL=0
MOVL C00884 V=800.0 PL=0
MOVL C00885 V=800.0 PL=0
MOVL C00886 V=800.0 PL=0
MOVL C00887 V=800.0 PL=0
MOVL C00888 V=800.0 PL=0
MOVL C00889 V=800.0 PL=0
MOVL C00890 V=800.0 PL=0
MOVL C00891 V=800.0 PL=0
MOVL C00892 V=800.0 PL=0
MOVL C00893 V=800.0 PL=0
MOVL C00894 V=800.0 PL=0
MOVL C00895 V=800.0 PL=0
MOVL C00896 V=800.0 PL=0
MOVL C00897 V=800.0 PL=0
MOVL C00898 V=800.0 PL=0
MOVL C00899 V=800.0 PL=0
MOVL C00900 V=800.0 PL=0
MOVL C00901 V=800.0 PL=0
MOVL C00902 V=800.0 PL=0
MOVL C00903 V=800.0 PL=0
MOVL C00904 V=800.0 PL=0
MOVL C00905 V=800.0 PL=0
MOVL C00906 V=800.0 PL=0
MOVL C00907 V=800.0 PL=0
MOVL C00908 V=800.0 PL=0
MOVL C00909 V=800.0 PL=0
MOVL C00910 V=800.0 PL=0
MOVL C00911 V=800.0 PL=0
MOVL C00912 V=800.0 PL=0
MOVL C00913 V=800.0 PL=0
MOVL C00914 V=800.0 PL=0
MOVL C00915 V=800.0 PL=0
MOVL C00916 V=800.0 PL=0
MOVL C00917 V=800.0 PL=0
MOVL C00918 V=800.0 PL=0
MOVL C00919 V=800.0 PL=0
MOVL C00920 V=800.0 PL=0
MOVL C00921 V=800.0 PL=0
MOVL C00922 V=800.0 PL=0
MOVL C00923 V=800.0 PL=0
MOVL C00924 V=800.0 PL=0
MOVL C00925 V=800.0 PL=0
MOVL C00926 V=800.0 PL=0
MOVL C00927 V=800.0 PL=0
MOVL C00928 V=800.0 PL=0
MOVL C00929 V=800.0 PL=0
MOVL C00930 V=800.0 PL=0
MOVL C00931 V=800.0 PL=0
MOVL C00932 V=800.0 PL=0
MOVL C00933 V=800.0 PL=0
MOVL C00934 V=800.0 PL=0
MOVL C00935 V=800.0 PL=0
MOVL C00936 V=800.0 PL=0
MOVL C00937 V=800.0 PL=0
MOVL C00938 V=800.0 PL=0
MOVL C00939 V=800.0 PL=0
MOVL C00940 V=800.0 PL=0
MOVL C00941 V=800.0 PL=0
MOVL C00942 V=800.0 PL=0
MOVL C00943 V=800.0 PL=0
MOVL C00944 V=800.0 PL=0
MOVL C00945 V=800.0 PL=0
MOVL C00946 V=800.0 PL=0
MOVL C00947 V=800.0 PL=0
MOVL C00948 V=800.0 PL=0
MOVL C00949 V=800.0 PL=0
MOVL C00950 V=800.0 PL=0
MOVL C00951 V=800.0 PL=0
MOVL C00952 V=800.0 PL=0
MOVL C00953 V=800.0 PL=0
MOVL C00954 V=800.0 PL=0
MOVL C00955 V=800.0 PL=0
MOVL C00956 V=800.0 PL=0
MOVL C00957 V=800.0 PL=0
MOVL C00958 V=800.0 PL=0
MOVL C00959 V=800.0 PL=0
MOVL C00960 V=800.0 PL=0
MOVL C00961 V=800.0 PL=0
MOVL C00962 V=800.0 PL=0
MOVL C00963 V=800.0 PL=0
MOVL C00964 V=800.0 PL=0
MOVL C00965 V=800.0 PL=0
MOVL C00966 V=800.0 PL=0
MOVL C00967 V=800.0 PL=0
MOVL C00968 V=800.0 PL=0
MOVL C00969 V=800.0 PL=0
MOVL C00970 V=800.0 PL=0
MOVL C00971 V=800.0 PL=0
MOVL C00972 V=800.0 PL=0
MOVL C00973 V=800.0 PL=0
MOVL C00974 V=800.0 PL=0
MOVL C00975 V=800.0 PL=0
MOVL C00976 V=800.0 PL=0
MOVL C00977 V=800.0 PL=0
MOVL C00978 V=800.0 PL=0
MOVL C00979 V=800.0 PL=0
MOVL C00980 V=800.0 PL=0
MOVL C00981 V=800.0 PL=0
MOVL C00982 V=800.0 PL=0
MOVL C00983 V=800.0 PL=0
MOVL C00984 V=800.0 PL=0
MOVL C00985 V=800.0 PL=0
MOVL C00986 V=800.0 PL=0
MOVL C00987 V=800.0 PL=0
MOVL C00988 V=800.0 PL=0
MOVL C00989 V=800.0 PL=0
MOVL C00990 V=800.0 PL=0
MOVL C00991 V=800.0 PL=0
MOVL C00992 V=800.0 PL=0
MOVL C00993 V=800.0 PL=0
MOVL C00994 V=800.0 PL=0
MOVL C00995 V=800.0 PL=0
MOVL C00996 V=800.0 PL=0
MOVL C00997 V=800.0 PL=0
MOVL C00998 V=800.0 PL=0
MOVL C00999 V=800.0 PL=0
MOVL C01000 V=800.0 PL=0
MOVL C01001 V=800.0 PL=0
MOVL C01002 V=800.0 PL=0
MOVL C01003 V=800.0 PL=0
MOVL C01004 V=800.0 PL=0
MOVL C01005 V=800.0 PL=0
MOVL C01006 V=800.0 PL=0
MOVL C01007 V=800.0 PL=0
MOVL C01008 V=800.0 PL=0
MOVL C01009 V=800.0 PL=0
MOVL C01010 V=800.0 PL=0
MOVL C01011 V=800.0 PL=0
MOVL C01012 V=800.0 PL=0
MOVL C01013 V=800.0 PL=0
MOVL C01014 V=800.0 PL=0
MOVL C01015 V=800.0 PL=0
MOVL C01016 V=800.0 PL=0
MOVL C01017 V=800.0 PL=0
MOVL C01018 V=800.0 PL=0
MOVL C01019 V=800.0 PL=0
MOVL C01020 V=800.0 PL=0
MOVL C01021 V=800.0 PL=0
MOVL C01022 V=800.0 PL=0
MOVL C01023 V=800.0 PL=0
MOVL C01024 V=800.0 PL=0
MOVL C01025 V=800.0 PL=0
MOVL C01026 V=800.0 PL=0
MOVL C01027 V=800.0 PL=0
MOVL C01028 V=800.0 PL=0
MOVL C01029 V=800.0 PL=0
MOVL C01030 V=800.0 PL=0
MOVL C01031 V=800.0 PL=0
MOVL C01032 V=800.0 PL=0
MOVL C01033 V=800.0 PL=0
MOVL C01034 V=800.0 PL=0
MOVL C01035 V=800.0 PL=0
MOVL C01036 V=800.0 PL=0
MOVL C01037 V=800.0 PL=0
MOVL C01038 V=800.0 PL=0
MOVL C01039 V=800.0 PL=0
MOVL C01040 V=800.0 PL=0
MOVL C01041 V=800.0 PL=0
MOVL C01042 V=800.0 PL=0
MOVL C01043 V=800.0 PL=0
MOVL C01044 V=800.0 PL=0
MOVL C01045 V=800.0 PL=0
MOVL C01046 V=800.0 PL=0
MOVL C01047 V=800.0 PL=0
MOVL C01048 V=800.0 PL=0
MOVL C01049 V=800.0 PL=0
MOVL C01050 V=800.0 PL=0
MOVL C01051 V=800.0 PL=0
MOVL C01052 V=800.0 PL=0
MOVL C01053 V=800.0 PL=0
MOVL C01054 V=800.0 PL=0
MOVL C01055 V=800.0 PL=0
MOVL C01056 V=800.0 PL=0
MOVL C01057 V=800.0 PL=0
MOVL C01058 V=800.0 PL=0
MOVL C01059 V=800.0 PL=0
MOVL C01060 V=800.0 PL=0
MOVL C01061 V=800.0 PL=0
MOVL C01062 V=800.0 PL=0
MOVL C01063 V=800.0 PL=0
MOVL C01064 V=800.0 PL=0
MOVL C01065 V=800.0 PL=0
MOVL C01066 V=800.0 PL=0
MOVL C01067 V=800.0 PL=0
MOVL C01068 V=800.0 PL=0
MOVL C01069 V=800.0 PL=0
MOVL C01070 V=800.0 PL=0
MOVL C01071 V=800.0 PL=0
MOVL C01072 V=800.0 PL=0
MOVL C01073 V=800.0 PL=0
MOVL C01074 V=800.0 PL=0
MOVL C01075 V=800.0 PL=0
MOVL C01076 V=800.0 PL=0
MOVL C01077 V=800.0 PL=0
MOVL C01078 V=800.0 PL=0
MOVL C01079 V=800.0 PL=0
MOVL C01080 V=800.0 PL=0
MOVL C01081 V=800.0 PL=0
MOVL C01082 V=800.0 PL=0
MOVL C01083 V=800.0 PL=0
MOVL C01084 V=800.0 PL=0
MOVL C01085 V=800.0 PL=0
MOVL C01086 V=800.0 PL=0
MOVL C01087 V=800.0 PL=0
MOVL C01088 V=800.0 PL=0
MOVL C01089 V=800.0 PL=0
MOVL C01090 V=800.0 PL=0
MOVL C01091 V=800.0 PL=0
MOVL C01092 V=800.0 PL=0
MOVL C01093 V=800.0 PL=0
MOVL C01094 V=800.0 PL=0
MOVL C01095 V=800.0 PL=0
MOVL C01096 V=800.0 PL=0
MOVL C01097 V=800.0 PL=0
MOVL C01098 V=800.0 PL=0
MOVL C01099 V=800.0 PL=0
MOVL C01100 V=800.0 PL=0
MOVL C01101 V=800.0 PL=0
MOVL C01102 V=800.0 PL=0
MOVL C01103 V=800.0 PL=0
MOVL C01104 V=800.0 PL=0
MOVL C01105 V=800.0 PL=0
MOVL C01106 V=800.0 PL=0
MOVL C01107 V=800.0 PL=0
MOVL C01108 V=800.0 PL=0
MOVL C01109 V=800.0 PL=0
MOVL C01110 V=800.0 PL=0
MOVL C01111 V=800.0 PL=0
MOVL C01112 V=800.0 PL=0
MOVL C01113 V=800.0 PL=0
MOVL C01114 V=800.0 PL=0
MOVL C01115 V=800.0 PL=0
MOVL C01116 V=800.0 PL=0
MOVL C01117 V=800.0 PL=0
MOVL C01118 V=800.0 PL=0
MOVL C01119 V=800.0 PL=0
MOVL C01120 V=800.0 PL=0
MOVL C01121 V=800.0 PL=0
MOVL C01122 V=800.0 PL=0
MOVL C01123 V=800.0 PL=0
MOVL C01124 V=800.0 PL=0
MOVL C01125 V=800.0 PL=0
MOVL C01126 V=800.0 PL=0
MOVL C01127 V=800.0 PL=0
MOVL C01128 V=800.0 PL=0
MOVL C01129 V=800.0 PL=0
MOVL C01130 V=800.0 PL=0
MOVL C01131 V=800.0 PL=0
MOVL C01132 V=800.0 PL=0
MOVL C01133 V=800.0 PL=0
MOVL C01134 V=800.0 PL=0
MOVL C01135 V=800.0 PL=0
MOVL C01136 V=800.0 PL=0
MOVL C01137 V=800.0 PL=0
MOVL C01138 V=800.0 PL=0
MOVL C01139 V=800.0 PL=0
MOVL C01140 V=800.0 PL=0
MOVL C01141 V=800.0 PL=0
MOVL C01142 V=800.0 PL=0
MOVL C01143 V=800.0 PL=0
MOVL C01144 V=800.0 PL=0
MOVL C01145 V=800.0 PL=0
MOVL C01146 V=800.0 PL=0
MOVL C01147 V=800.0 PL=0
MOVL C01148 V=800.0 PL=0
MOVL C01149 V=800.0 PL=0
MOVL C01150 V=800.0 PL=0
MOVL C01151 V=800.0 PL=0
MOVL C01152 V=800.0 PL=0
MOVL C01153 V=800.0 PL=0
MOVL C01154 V=800.0 PL=0
MOVL C01155 V=800.0 PL=0
MOVL C01156 V=800.0 PL=0
MOVL C01157 V=800.0 PL=0
MOVL C01158 V=800.0 PL=0
MOVL C01159 V=800.0 PL=0
MOVL C01160 V=800.0 PL=0
MOVL C01161 V=800.0 PL=0
MOVL C01162 V=800.0 PL=0
MOVL C01163 V=800.0 PL=0
MOVL C01164 V=800.0 PL=0
MOVL C01165 V=800.0 PL=0
MOVL C01166 V=800.0 PL=0
MOVL C01167 V=800.0 PL=0
MOVL C01168 V=800.0 PL=0
MOVL C01169 V=800.0 PL=0
MOVL C01170 V=800.0 PL=0
MOVL C01171 V=800.0 PL=0
MOVL C01172 V=800.0 PL=0
MOVL C01173 V=800.0 PL=0
MOVL C01174 V=800.0 PL=0
MOVL C01175 V=800.0 PL=0
MOVL C01176 V=800.0 PL=0
MOVL C01177 V=800.0 PL=0
MOVL C01178 V=800.0 PL=0
MOVL C01179 V=800.0 PL=0
MOVL C01180 V=800.0 PL=0
MOVL C01181 V=800.0 PL=0
MOVL C01182 V=800.0 PL=0
MOVL C01183 V=800.0 PL=0
MOVL C01184 V=800.0 PL=0
MOVL C01185 V=800.0 PL=0
MOVL C01186 V=800.0 PL=0
MOVL C01187 V=800.0 PL=0
MOVL C01188 V=800.0 PL=0
MOVL C01189 V=800.0 PL=0
MOVL C01190 V=800.0 PL=0
MOVL C01191 V=800.0 PL=0
MOVL C01192 V=800.0 PL=0
MOVL C01193 V=800.0 PL=0
MOVL C01194 V=800.0 PL=0
MOVL C01195 V=800.0 PL=0
MOVL C01196 V=800.0 PL=0
MOVL C01197 V=800.0 PL=0
MOVL C01198 V=800.0 PL=0
MOVL C01199 V=800.0 PL=0
MOVL C01200 V=800.0 PL=0
MOVL C01201 V=800.0 PL=0
MOVL C01202 V=800.0 PL=0
MOVL C01203 V=800.0 PL=0
MOVL C01204 V=800.0 PL=0
MOVL C01205 V=800.0 PL=0
MOVL C01206 V=800.0 PL=0
MOVL C01207 V=800.0 PL=0
MOVL C01208 V=800.0 PL=0
MOVL C01209 V=800.0 PL=0
MOVL C01210 V=800.0 PL=0
MOVL C01211 V=800.0 PL=0
MOVL C01212 V=800.0 PL=0
MOVL C01213 V=800.0 PL=0
MOVL C01214 V=800.0 PL=0
MOVL C01215 V=800.0 PL=0
MOVL C01216 V=800.0 PL=0
MOVL C01217 V=800.0 PL=0
MOVL C01218 V=800.0 PL=0
MOVL C01219 V=800.0 PL=0
MOVL C01220 V=800.0 PL=0
MOVL C01221 V=800.0 PL=0
MOVL C01222 V=800.0 PL=0
MOVL C01223 V=800.0 PL=0
MOVL C01224 V=800.0 PL=0
MOVL C01225 V=800.0 PL=0
MOVL C01226 V=800.0 PL=0
MOVL C01227 V=800.0 PL=0
MOVL C01228 V=800.0 PL=0
MOVL C01229 V=800.0 PL=0
MOVL C01230 V=800.0 PL=0
MOVL C01231 V=800.0 PL=0
MOVL C01232 V=800.0 PL=0
MOVL C01233 V=800.0 PL=0
MOVL C01234 V=800.0 PL=0
MOVL C01235 V=800.0 PL=0
MOVL C01236 V=800.0 PL=0
MOVL C01237 V=800.0 PL=0
MOVL C01238 V=800.0 PL=0
MOVL C01239 V=800.0 PL=0
MOVL C01240 V=800.0 PL=0
MOVL C01241 V=800.0 PL=0
MOVL C01242 V=800.0 PL=0
MOVL C01243 V=800.0 PL=0
MOVL C01244 V=800.0 PL=0
MOVL C01245 V=800.0 PL=0
MOVL C01246 V=800.0 PL=0
MOVL C01247 V=800.0 PL=0
MOVL C01248 V=800.0 PL=0
MOVL C01249 V=800.0 PL=0
MOVL C01250 V=800.0 PL=0
MOVL C01251 V=800.0 PL=0
MOVL C01252 V=800.0 PL=0
MOVL C01253 V=800.0 PL=0
MOVL C01254 V=800.0 PL=0
MOVL C01255 V=800.0 PL=0
MOVL C01256 V=800.0 PL=0
MOVL C01257 V=800.0 PL=0
MOVL C01258 V=800.0 PL=0
MOVL C01259 V=800.0 PL=0
MOVL C01260 V=800.0 PL=0
MOVL C01261 V=800.0 PL=0
MOVL C01262 V=800.0 PL=0
MOVL C01263 V=800.0 PL=0
MOVL C01264 V=800.0 PL=0
MOVL C01265 V=800.0 PL=0
MOVL C01266 V=800.0 PL=0
MOVL C01267 V=800.0 PL=0
MOVL C01268 V=800.0 PL=0
MOVL C01269 V=800.0 PL=0
MOVL C01270 V=800.0 PL=0
MOVL C01271 V=800.0 PL=0
MOVL C01272 V=800.0 PL=0
MOVL C01273 V=800.0 PL=0
MOVL C01274 V=800.0 PL=0
MOVL C01275 V=800.0 PL=0
MOVL C01276 V=800.0 PL=0
MOVL C01277 V=800.0 PL=0
MOVL C01278 V=800.0 PL=0
MOVL C01279 V=800.0 PL=0
MOVL C01280 V=800.0 PL=0
MOVL C01281 V=800.0 PL=0
MOVL C01282 V=800.0 PL=0
MOVL C01283 V=800.0 PL=0
MOVL C01284 V=800.0 PL=0
MOVL C01285 V=800.0 PL=0
MOVL C01286 V=800.0 PL=0
MOVL C01287 V=800.0 PL=0
MOVL C01288 V=800.0 PL=0
MOVL C01289 V=800.0 PL=0
MOVL C01290 V=800.0 PL=0
MOVL C01291 V=800.0 PL=0
MOVL C01292 V=800.0 PL=0
MOVL C01293 V=800.0 PL=0
MOVL C01294 V=800.0 PL=0
MOVL C01295 V=800.0 PL=0
MOVL C01296 V=800.0 PL=0
MOVL C01297 V=800.0 PL=0
MOVL C01298 V=800.0 PL=0
MOVL C01299 V=800.0 PL=0
MOVL C01300 V=800.0 PL=0
MOVL C01301 V=800.0 PL=0
MOVL C01302 V=800.0 PL=0
MOVL C01303 V=800.0 PL=0
MOVL C01304 V=800.0 PL=0
MOVL C01305 V=800.0 PL=0
MOVL C01306 V=800.0 PL=0
MOVL C01307 V=800.0 PL=0
MOVL C01308 V=800.0 PL=0
MOVL C01309 V=800.0 PL=0
MOVL C01310 V=800.0 PL=0
MOVL C01311 V=800.0 PL=0
MOVL C01312 V=800.0 PL=0
MOVL C01313 V=800.0 PL=0
MOVL C01314 V=800.0 PL=0
MOVL C01315 V=800.0 PL=0
MOVL C01316 V=800.0 PL=0
MOVL C01317 V=800.0 PL=0
MOVL C01318 V=800.0 PL=0
MOVL C01319 V=800.0 PL=0
MOVL C01320 V=800.0 PL=0
MOVL C01321 V=800.0 PL=0
MOVL C01322 V=800.0 PL=0
MOVL C01323 V=800.0 PL=0
MOVL C01324 V=800.0 PL=0
MOVL C01325 V=800.0 PL=0
MOVL C01326 V=800.0 PL=0
MOVL C01327 V=800.0 PL=0
MOVL C01328 V=800.0 PL=0
MOVL C01329 V=800.0 PL=0
MOVL C01330 V=800.0 PL=0
MOVL C01331 V=800.0 PL=0
MOVL C01332 V=800.0 PL=0
MOVL C01333 V=800.0 PL=0
MOVL C01334 V=800.0 PL=0
MOVL C01335 V=800.0 PL=0
MOVL C01336 V=800.0 PL=0
MOVL C01337 V=800.0 PL=0
MOVL C01338 V=800.0 PL=0
MOVL C01339 V=800.0 PL=0
MOVL C01340 V=800.0 PL=0
MOVL C01341 V=800.0 PL=0
MOVL C01342 V=800.0 PL=0
MOVL C01343 V=800.0 PL=0
MOVL C01344 V=800.0 PL=0
MOVL C01345 V=800.0 PL=0
MOVL C01346 V=800.0 PL=0
MOVL C01347 V=800.0 PL=0
MOVL C01348 V=800.0 PL=0
MOVL C01349 V=800.0 PL=0
MOVL C01350 V=800.0 PL=0
MOVL C01351 V=800.0 PL=0
MOVL C01352 V=800.0 PL=0
MOVL C01353 V=800.0 PL=0
MOVL C01354 V=800.0 PL=0
MOVL C01355 V=800.0 PL=0
MOVL C01356 V=800.0 PL=0
MOVL C01357 V=800.0 PL=0
MOVL C01358 V=800.0 PL=0
MOVL C01359 V=800.0 PL=0
MOVL C01360 V=800.0 PL=0
MOVL C01361 V=800.0 PL=0
MOVL C01362 V=800.0 PL=0
MOVL C01363 V=800.0 PL=0
MOVL C01364 V=800.0 PL=0
MOVL C01365 V=800.0 PL=0
MOVL C01366 V=800.0 PL=0
MOVL C01367 V=800.0 PL=0
MOVL C01368 V=800.0 PL=0
MOVL C01369 V=800.0 PL=0
MOVL C01370 V=800.0 PL=0
MOVL C01371 V=800.0 PL=0
MOVL C01372 V=800.0 PL=0
MOVL C01373 V=800.0 PL=0
MOVL C01374 V=800.0 PL=0
MOVL C01375 V=800.0 PL=0
MOVL C01376 V=800.0 PL=0
MOVL C01377 V=800.0 PL=0
MOVL C01378 V=800.0 PL=0
MOVL C01379 V=800.0 PL=0
MOVL C01380 V=800.0 PL=0
MOVL C01381 V=800.0 PL=0
MOVL C01382 V=800.0 PL=0
MOVL C01383 V=800.0 PL=0
MOVL C01384 V=800.0 PL=0
MOVL C01385 V=800.0 PL=0
MOVL C01386 V=800.0 PL=0
MOVL C01387 V=800.0 PL=0
MOVL C01388 V=800.0 PL=0
MOVL C01389 V=800.0 PL=0
MOVL C01390 V=800.0 PL=0
MOVL C01391 V=800.0 PL=0
MOVL C01392 V=800.0 PL=0
MOVL C01393 V=800.0 PL=0
MOVL C01394 V=800.0 PL=0
MOVL C01395 V=800.0 PL=0
MOVL C01396 V=800.0 PL=0
MOVL C01397 V=800.0 PL=0
MOVL C01398 V=800.0 PL=0
MOVL C01399 V=800.0 PL=0
MOVL C01400 V=800.0 PL=0
MOVL C01401 V=800.0 PL=0
MOVL C01402 V=800.0 PL=0
MOVL C01403 V=800.0 PL=0
MOVL C01404 V=800.0 PL=0
MOVL C01405 V=800.0 PL=0
MOVL C01406 V=800.0 PL=0
MOVL C01407 V=800.0 PL=0
MOVL C01408 V=800.0 PL=0
MOVL C01409 V=800.0 PL=0
MOVL C01410 V=800.0 PL=0
MOVL C01411 V=800.0 PL=0
MOVL C01412 V=800.0 PL=0
MOVL C01413 V=800.0 PL=0
MOVL C01414 V=800.0 PL=0
MOVL C01415 V=800.0 PL=0
MOVL C01416 V=800.0 PL=0
MOVL C01417 V=800.0 PL=0
MOVL C01418 V=800.0 PL=0
MOVL C01419 V=800.0 PL=0
MOVL C01420 V=800.0 PL=0
MOVL C01421 V=800.0 PL=0
MOVL C01422 V=800.0 PL=0
MOVL C01423 V=800.0 PL=0
MOVL C01424 V=800.0 PL=0
MOVL C01425 V=800.0 PL=0
MOVL C01426 V=800.0 PL=0
MOVL C01427 V=800.0 PL=0
MOVL C01428 V=800.0 PL=0
MOVL C01429 V=800.0 PL=0
MOVL C01430 V=800.0 PL=0
MOVL C01431 V=800.0 PL=0
MOVL C01432 V=800.0 PL=0
MOVL C01433 V=800.0 PL=0
MOVL C01434 V=800.0 PL=0
MOVL C01435 V=800.0 PL=0
MOVL C01436 V=800.0 PL=0
MOVL C01437 V=800.0 PL=0
MOVL C01438 V=800.0 PL=0
MOVL C01439 V=800.0 PL=0
MOVL C01440 V=800.0 PL=0
MOVL C01441 V=800.0 PL=0
MOVL C01442 V=800.0 PL=0
MOVL C01443 V=800.0 PL=0
MOVL C01444 V=800.0 PL=0
MOVL C01445 V=800.0 PL=0
MOVL C01446 V=800.0 PL=0
MOVL C01447 V=800.0 PL=0
MOVL C01448 V=800.0 PL=0
MOVL C01449 V=800.0 PL=0
MOVL C01450 V=800.0 PL=0
MOVL C01451 V=800.0 PL=0
MOVL C01452 V=800.0 PL=0
MOVL C01453 V=800.0 PL=0
MOVL C01454 V=800.0 PL=0
MOVL C01455 V=800.0 PL=0
MOVL C01456 V=800.0 PL=0
MOVL C01457 V=800.0 PL=0
MOVL C01458 V=800.0 PL=0
MOVL C01459 V=800.0 PL=0
MOVL C01460 V=800.0 PL=0
MOVL C01461 V=800.0 PL=0
MOVL C01462 V=800.0 PL=0
MOVL C01463 V=800.0 PL=0
MOVL C01464 V=800.0 PL=0
MOVL C01465 V=800.0 PL=0
MOVL C01466 V=800.0 PL=0
MOVL C01467 V=800.0 PL=0
MOVL C01468 V=800.0 PL=0
MOVL C01469 V=800.0 PL=0
MOVL C01470 V=800.0 PL=0
MOVL C01471 V=800.0 PL=0
MOVL C01472 V=800.0 PL=0
MOVL C01473 V=800.0 PL=0
MOVL C01474 V=800.0 PL=0
MOVL C01475 V=800.0 PL=0
MOVL C01476 V=800.0 PL=0
MOVL C01477 V=800.0 PL=0
MOVL C01478 V=800.0 PL=0
MOVL C01479 V=800.0 PL=0
MOVL C01480 V=800.0 PL=0
MOVL C01481 V=800.0 PL=0
MOVL C01482 V=800.0 PL=0
MOVL C01483 V=800.0 PL=0
MOVL C01484 V=800.0 PL=0
MOVL C01485 V=800.0 PL=0
MOVL C01486 V=800.0 PL=0
MOVL C01487 V=800.0 PL=0
MOVL C01488 V=800.0 PL=0
MOVL C01489 V=800.0 PL=0
MOVL C01490 V=800.0 PL=0
MOVL C01491 V=800.0 PL=0
MOVL C01492 V=800.0 PL=0
MOVL C01493 V=800.0 PL=0
MOVL C01494 V=800.0 PL=0
MOVL C01495 V=800.0 PL=0
MOVL C01496 V=800.0 PL=0
MOVL C01497 V=800.0 PL=0
MOVL C01498 V=800.0 PL=0
MOVL C01499 V=800.0 PL=0
MOVL C01500 V=800.0 PL=0
MOVL C01501 V=800.0 PL=0
MOVL C01502 V=800.0 PL=0
MOVL C01503 V=800.0 PL=0
MOVL C01504 V=800.0 PL=0
MOVL C01505 V=800.0 PL=0
MOVL C01506 V=800.0 PL=0
MOVL C01507 V=800.0 PL=0
MOVL C01508 V=800.0 PL=0
MOVL C01509 V=800.0 PL=0
MOVL C01510 V=800.0 PL=0
MOVL C01511 V=800.0 PL=0
MOVL C01512 V=800.0 PL=0
MOVL C01513 V=800.0 PL=0
MOVL C01514 V=800.0 PL=0
MOVL C01515 V=800.0 PL=0
MOVL C01516 V=800.0 PL=0
MOVL C01517 V=800.0 PL=0
MOVL C01518 V=800.0 PL=0
MOVL C01519 V=800.0 PL=0
MOVL C01520 V=800.0 PL=0
MOVL C01521 V=800.0 PL=0
MOVL C01522 V=800.0 PL=0
MOVL C01523 V=800.0 PL=0
MOVL C01524 V=800.0 PL=0
MOVL C01525 V=800.0 PL=0
MOVL C01526 V=800.0 PL=0
MOVL C01527 V=800.0 PL=0
MOVL C01528 V=800.0 PL=0
MOVL C01529 V=800.0 PL=0
MOVL C01530 V=800.0 PL=0
MOVL C01531 V=800.0 PL=0
MOVL C01532 V=800.0 PL=0
MOVL C01533 V=800.0 PL=0
MOVL C01534 V=800.0 PL=0
MOVL C01535 V=800.0 PL=0
MOVL C01536 V=800.0 PL=0
MOVL C01537 V=800.0 PL=0
MOVL C01538 V=800.0 PL=0
MOVL C01539 V=800.0 PL=0
MOVL C01540 V=800.0 PL=0
MOVL C01541 V=800.0 PL=0
MOVL C01542 V=800.0 PL=0
MOVL C01543 V=800.0 PL=0
MOVL C01544 V=800.0 PL=0
MOVL C01545 V=800.0 PL=0
MOVL C01546 V=800.0 PL=0
MOVL C01547 V=800.0 PL=0
MOVL C01548 V=800.0 PL=0
MOVL C01549 V=800.0 PL=0
MOVL C01550 V=800.0 PL=0
MOVL C01551 V=800.0 PL=0
MOVL C01552 V=800.0 PL=0
MOVL C01553 V=800.0 PL=0
MOVL C01554 V=800.0 PL=0
MOVL C01555 V=800.0 PL=0
MOVL C01556 V=800.0 PL=0
MOVL C01557 V=800.0 PL=0
MOVL C01558 V=800.0 PL=0
MOVL C01559 V=800.0 PL=0
MOVL C01560 V=800.0 PL=0
MOVL C01561 V=800.0 PL=0
MOVL C01562 V=800.0 PL=0
MOVL C01563 V=800.0 PL=0
MOVL C01564 V=800.0 PL=0
MOVL C01565 V=800.0 PL=0
MOVL C01566 V=800.0 PL=0
MOVL C01567 V=800.0 PL=0
MOVL C01568 V=800.0 PL=0
MOVL C01569 V=800.0 PL=0
MOVL C01570 V=800.0 PL=0
MOVL C01571 V=800.0 PL=0
MOVL C01572 V=800.0 PL=0
MOVL C01573 V=800.0 PL=0
MOVL C01574 V=800.0 PL=0
MOVL C01575 V=800.0 PL=0
MOVL C01576 V=800.0 PL=0
MOVL C01577 V=800.0 PL=0
MOVL C01578 V=800.0 PL=0
MOVL C01579 V=800.0 PL=0
MOVL C01580 V=800.0 PL=0
MOVL C01581 V=800.0 PL=0
MOVL C01582 V=800.0 PL=0
MOVL C01583 V=800.0 PL=0
MOVL C01584 V=800.0 PL=0
MOVL C01585 V=800.0 PL=0
MOVL C01586 V=800.0 PL=0
MOVL C01587 V=800.0 PL=0
MOVL C01588 V=800.0 PL=0
MOVL C01589 V=800.0 PL=0
MOVL C01590 V=800.0 PL=0
MOVL C01591 V=800.0 PL=0
MOVL C01592 V=800.0 PL=0
MOVL C01593 V=800.0 PL=0
MOVL C01594 V=800.0 PL=0
MOVL C01595 V=800.0 PL=0
MOVL C01596 V=800.0 PL=0
MOVL C01597 V=800.0 PL=0
MOVL C01598 V=800.0 PL=0
MOVL C01599 V=800.0 PL=0
MOVL C01600 V=800.0 PL=0
MOVL C01601 V=800.0 PL=0
MOVL C01602 V=800.0 PL=0
MOVL C01603 V=800.0 PL=0
MOVL C01604 V=800.0 PL=0
MOVL C01605 V=800.0 PL=0
MOVL C01606 V=800.0 PL=0
MOVL C01607 V=800.0 PL=0
MOVL C01608 V=800.0 PL=0
MOVL C01609 V=800.0 PL=0
MOVL C01610 V=800.0 PL=0
MOVL C01611 V=800.0 PL=0
MOVL C01612 V=800.0 PL=0
MOVL C01613 V=800.0 PL=0
MOVL C01614 V=800.0 PL=0
MOVL C01615 V=800.0 PL=0
MOVL C01616 V=800.0 PL=0
MOVL C01617 V=800.0 PL=0
MOVL C01618 V=800.0 PL=0
MOVL C01619 V=800.0 PL=0
MOVL C01620 V=800.0 PL=0
MOVL C01621 V=800.0 PL=0
MOVL C01622 V=800.0 PL=0
MOVL C01623 V=800.0 PL=0
MOVL C01624 V=800.0 PL=0
MOVL C01625 V=800.0 PL=0
MOVL C01626 V=800.0 PL=0
MOVL C01627 V=800.0 PL=0
MOVL C01628 V=800.0 PL=0
MOVL C01629 V=800.0 PL=0
MOVL C01630 V=800.0 PL=0
MOVL C01631 V=800.0 PL=0
MOVL C01632 V=800.0 PL=0
MOVL C01633 V=800.0 PL=0
MOVL C01634 V=800.0 PL=0
MOVL C01635 V=800.0 PL=0
MOVL C01636 V=800.0 PL=0
MOVL C01637 V=800.0 PL=0
MOVL C01638 V=800.0 PL=0
MOVL C01639 V=800.0 PL=0
MOVL C01640 V=800.0 PL=0
MOVL C01641 V=800.0 PL=0
MOVL C01642 V=800.0 PL=0
MOVL C01643 V=800.0 PL=0
MOVL C01644 V=800.0 PL=0
MOVL C01645 V=800.0 PL=0
MOVL C01646 V=800.0 PL=0
MOVL C01647 V=800.0 PL=0
MOVL C01648 V=800.0 PL=0
MOVL C01649 V=800.0 PL=0
MOVL C01650 V=800.0 PL=0
MOVL C01651 V=800.0 PL=0
MOVL C01652 V=800.0 PL=0
MOVL C01653 V=800.0 PL=0
MOVL C01654 V=800.0 PL=0
MOVL C01655 V=800.0 PL=0
MOVL C01656 V=800.0 PL=0
MOVL C01657 V=800.0 PL=0
MOVL C01658 V=800.0 PL=0
MOVL C01659 V=800.0 PL=0
MOVL C01660 V=800.0 PL=0
MOVL C01661 V=800.0 PL=0
MOVL C01662 V=800.0 PL=0
MOVL C01663 V=800.0 PL=0
MOVL C01664 V=800.0 PL=0
MOVL C01665 V=800.0 PL=0
MOVL C01666 V=800.0 PL=0
MOVL C01667 V=800.0 PL=0
MOVL C01668 V=800.0 PL=0
MOVL C01669 V=800.0 PL=0
MOVL C01670 V=800.0 PL=0
MOVL C01671 V=800.0 PL=0
MOVL C01672 V=800.0 PL=0
MOVL C01673 V=800.0 PL=0
MOVL C01674 V=800.0 PL=0
MOVL C01675 V=800.0 PL=0
MOVL C01676 V=800.0 PL=0
MOVL C01677 V=800.0 PL=0
MOVL C01678 V=800.0 PL=0
MOVL C01679 V=800.0 PL=0
MOVL C01680 V=800.0 PL=0
MOVL C01681 V=800.0 PL=0
MOVL C01682 V=800.0 PL=0
MOVL C01683 V=800.0 PL=0
MOVL C01684 V=800.0 PL=0
MOVL C01685 V=800.0 PL=0
MOVL C01686 V=800.0 PL=0
MOVL C01687 V=800.0 PL=0
MOVL C01688 V=800.0 PL=0
MOVL C01689 V=800.0 PL=0
MOVL C01690 V=800.0 PL=0
MOVL C01691 V=800.0 PL=0
MOVL C01692 V=800.0 PL=0
MOVL C01693 V=800.0 PL=0
MOVL C01694 V=800.0 PL=0
MOVL C01695 V=800.0 PL=0
MOVL C01696 V=800.0 PL=0
MOVL C01697 V=800.0 PL=0
MOVL C01698 V=800.0 PL=0
MOVL C01699 V=800.0 PL=0
MOVL C01700 V=800.0 PL=0
MOVL C01701 V=800.0 PL=0
MOVL C01702 V=800.0 PL=0
MOVL C01703 V=800.0 PL=0
MOVL C01704 V=800.0 PL=0
MOVL C01705 V=800.0 PL=0
MOVL C01706 V=800.0 PL=0
MOVL C01707 V=800.0 PL=0
MOVL C01708 V=800.0 PL=0
MOVL C01709 V=800.0 PL=0
MOVL C01710 V=800.0 PL=0
MOVL C01711 V=800.0 PL=0
MOVL C01712 V=800.0 PL=0
MOVL C01713 V=800.0 PL=0
MOVL C01714 V=800.0 PL=0
MOVL C01715 V=800.0 PL=0
MOVL C01716 V=800.0 PL=0
MOVL C01717 V=800.0 PL=0
MOVL C01718 V=800.0 PL=0
MOVL C01719 V=800.0 PL=0
MOVL C01720 V=800.0 PL=0
MOVL C01721 V=800.0 PL=0
MOVL C01722 V=800.0 PL=0
MOVL C01723 V=800.0 PL=0
MOVL C01724 V=800.0 PL=0
MOVL C01725 V=800.0 PL=0
MOVL C01726 V=800.0 PL=0
MOVL C01727 V=800.0 PL=0
MOVL C01728 V=800.0 PL=0
MOVL C01729 V=800.0 PL=0
MOVL C01730 V=800.0 PL=0
MOVL C01731 V=800.0 PL=0
MOVL C01732 V=800.0 PL=0
MOVL C01733 V=800.0 PL=0
MOVL C01734 V=800.0 PL=0
MOVL C01735 V=800.0 PL=0
MOVL C01736 V=800.0 PL=0
MOVL C01737 V=800.0 PL=0
MOVL C01738 V=800.0 PL=0
MOVL C01739 V=800.0 PL=0
MOVL C01740 V=800.0 PL=0
MOVL C01741 V=800.0 PL=0
MOVL C01742 V=800.0 PL=0
MOVL C01743 V=800.0 PL=0
MOVL C01744 V=800.0 PL=0
MOVL C01745 V=800.0 PL=0
MOVL C01746 V=800.0 PL=0
MOVL C01747 V=800.0 PL=0
MOVL C01748 V=800.0 PL=0
MOVL C01749 V=800.0 PL=0
MOVL C01750 V=800.0 PL=0
MOVL C01751 V=800.0 PL=0
MOVL C01752 V=800.0 PL=0
MOVL C01753 V=800.0 PL=0
MOVL C01754 V=800.0 PL=0
MOVL C01755 V=800.0 PL=0
MOVL C01756 V=800.0 PL=0
MOVL C01757 V=800.0 PL=0
MOVL C01758 V=800.0 PL=0
MOVL C01759 V=800.0 PL=0
MOVL C01760 V=800.0 PL=0
MOVL C01761 V=800.0 PL=0
MOVL C01762 V=800.0 PL=0
MOVL C01763 V=800.0 PL=0
MOVL C01764 V=800.0 PL=0
MOVL C01765 V=800.0 PL=0
MOVL C01766 V=800.0 PL=0
MOVL C01767 V=800.0 PL=0
MOVL C01768 V=800.0 PL=0
MOVL C01769 V=800.0 PL=0
MOVL C01770 V=800.0 PL=0
MOVL C01771 V=800.0 PL=0
MOVL C01772 V=800.0 PL=0
MOVL C01773 V=800.0 PL=0
MOVL C01774 V=800.0 PL=0
MOVL C01775 V=800.0 PL=0
MOVL C01776 V=800.0 PL=0
MOVL C01777 V=800.0 PL=0
MOVL C01778 V=800.0 PL=0
MOVL C01779 V=800.0 PL=0
MOVL C01780 V=800.0 PL=0
MOVL C01781 V=800.0 PL=0
MOVL C01782 V=800.0 PL=0
MOVL C01783 V=800.0 PL=0
MOVL C01784 V=800.0 PL=0
MOVL C01785 V=800.0 PL=0
MOVL C01786 V=800.0 PL=0
MOVL C01787 V=800.0 PL=0
MOVL C01788 V=800.0 PL=0
MOVL C01789 V=800.0 PL=0
MOVL C01790 V=800.0 PL=0
MOVL C01791 V=800.0 PL=0
MOVL C01792 V=800.0 PL=0
MOVL C01793 V=800.0 PL=0
MOVL C01794 V=800.0 PL=0
MOVL C01795 V=800.0 PL=0
MOVL C01796 V=800.0 PL=0
MOVL C01797 V=800.0 PL=0
MOVL C01798 V=800.0 PL=0
MOVL C01799 V=800.0 PL=0
MOVL C01800 V=800.0 PL=0
MOVL C01801 V=800.0 PL=0
MOVL C01802 V=800.0 PL=0
MOVL C01803 V=800.0 PL=0
MOVL C01804 V=800.0 PL=0
MOVL C01805 V=800.0 PL=0
MOVL C01806 V=800.0 PL=0
MOVL C01807 V=800.0 PL=0
MOVL C01808 V=800.0 PL=0
MOVL C01809 V=800.0 PL=0
MOVL C01810 V=800.0 PL=0
MOVL C01811 V=800.0 PL=0
MOVL C01812 V=800.0 PL=0
MOVL C01813 V=800.0 PL=0
MOVL C01814 V=800.0 PL=0
MOVL C01815 V=800.0 PL=0
MOVL C01816 V=800.0 PL=0
MOVL C01817 V=800.0 PL=0
MOVL C01818 V=800.0 PL=0
MOVL C01819 V=800.0 PL=0
MOVL C01820 V=800.0 PL=0
MOVL C01821 V=800.0 PL=0
MOVL C01822 V=800.0 PL=0
MOVL C01823 V=800.0 PL=0
MOVL C01824 V=800.0 PL=0
MOVL C01825 V=800.0 PL=0
MOVL C01826 V=800.0 PL=0
MOVL C01827 V=800.0 PL=0
MOVL C01828 V=800.0 PL=0
MOVL C01829 V=800.0 PL=0
MOVL C01830 V=800.0 PL=0
MOVL C01831 V=800.0 PL=0
MOVL C01832 V=800.0 PL=0
MOVL C01833 V=800.0 PL=0
MOVL C01834 V=800.0 PL=0
MOVL C01835 V=800.0 PL=0
MOVL C01836 V=800.0 PL=0
MOVL C01837 V=800.0 PL=0
MOVL C01838 V=800.0 PL=0
MOVL C01839 V=800.0 PL=0
MOVL C01840 V=800.0 PL=0
MOVL C01841 V=800.0 PL=0
MOVL C01842 V=800.0 PL=0
MOVL C01843 V=800.0 PL=0
MOVL C01844 V=800.0 PL=0
MOVL C01845 V=800.0 PL=0
MOVL C01846 V=800.0 PL=0
MOVL C01847 V=800.0 PL=0
MOVL C01848 V=800.0 PL=0
MOVL C01849 V=800.0 PL=0
MOVL C01850 V=800.0 PL=0
MOVL C01851 V=800.0 PL=0
MOVL C01852 V=800.0 PL=0
MOVL C01853 V=800.0 PL=0
MOVL C01854 V=800.0 PL=0
MOVL C01855 V=800.0 PL=0
MOVL C01856 V=800.0 PL=0
MOVL C01857 V=800.0 PL=0
MOVL C01858 V=800.0 PL=0
MOVL C01859 V=800.0 PL=0
MOVL C01860 V=800.0 PL=0
MOVL C01861 V=800.0 PL=0
MOVL C01862 V=800.0 PL=0
MOVL C01863 V=800.0 PL=0
MOVL C01864 V=800.0 PL=0
MOVL C01865 V=800.0 PL=0
MOVL C01866 V=800.0 PL=0
MOVL C01867 V=800.0 PL=0
MOVL C01868 V=800.0 PL=0
MOVL C01869 V=800.0 PL=0
MOVL C01870 V=800.0 PL=0
MOVL C01871 V=800.0 PL=0
MOVL C01872 V=800.0 PL=0
MOVL C01873 V=800.0 PL=0
MOVL C01874 V=800.0 PL=0
MOVL C01875 V=800.0 PL=0
MOVL C01876 V=800.0 PL=0
MOVL C01877 V=800.0 PL=0
MOVL C01878 V=800.0 PL=0
MOVL C01879 V=800.0 PL=0
MOVL C01880 V=800.0 PL=0
MOVL C01881 V=800.0 PL=0
MOVL C01882 V=800.0 PL=0
MOVL C01883 V=800.0 PL=0
MOVL C01884 V=800.0 PL=0
MOVL C01885 V=800.0 PL=0
MOVL C01886 V=800.0 PL=0
MOVL C01887 V=800.0 PL=0
MOVL C01888 V=800.0 PL=0
MOVL C01889 V=800.0 PL=0
MOVL C01890 V=800.0 PL=0
MOVL C01891 V=800.0 PL=0
MOVL C01892 V=800.0 PL=0
MOVL C01893 V=800.0 PL=0
MOVL C01894 V=800.0 PL=0
MOVL C01895 V=800.0 PL=0
MOVL C01896 V=800.0 PL=0
MOVL C01897 V=800.0 PL=0
MOVL C01898 V=800.0 PL=0
MOVL C01899 V=800.0 PL=0
MOVL C01900 V=800.0 PL=0
MOVL C01901 V=800.0 PL=0
MOVL C01902 V=800.0 PL=0
MOVL C01903 V=800.0 PL=0
MOVL C01904 V=800.0 PL=0
MOVL C01905 V=800.0 PL=0
MOVL C01906 V=800.0 PL=0
MOVL C01907 V=800.0 PL=0
MOVL C01908 V=800.0 PL=0
MOVL C01909 V=800.0 PL=0
MOVL C01910 V=800.0 PL=0
MOVL C01911 V=800.0 PL=0
MOVL C01912 V=800.0 PL=0
MOVL C01913 V=800.0 PL=0
MOVL C01914 V=800.0 PL=0
MOVL C01915 V=800.0 PL=0
MOVL C01916 V=800.0 PL=0
MOVL C01917 V=800.0 PL=0
MOVL C01918 V=800.0 PL=0
MOVL C01919 V=800.0 PL=0
MOVL C01920 V=800.0 PL=0
MOVL C01921 V=800.0 PL=0
MOVL C01922 V=800.0 PL=0
MOVL C01923 V=800.0 PL=0
MOVL C01924 V=800.0 PL=0
MOVL C01925 V=800.0 PL=0
MOVL C01926 V=800.0 PL=0
MOVL C01927 V=800.0 PL=0
MOVL C01928 V=800.0 PL=0
MOVL C01929 V=800.0 PL=0
MOVL C01930 V=800.0 PL=0
MOVL C01931 V=800.0 PL=0
MOVL C01932 V=800.0 PL=0
MOVL C01933 V=800.0 PL=0
MOVL C01934 V=800.0 PL=0
MOVL C01935 V=800.0 PL=0
MOVL C01936 V=800.0 PL=0
MOVL C01937 V=800.0 PL=0
MOVL C01938 V=800.0 PL=0
MOVL C01939 V=800.0 PL=0
MOVL C01940 V=800.0 PL=0
MOVL C01941 V=800.0 PL=0
MOVL C01942 V=800.0 PL=0
MOVL C01943 V=800.0 PL=0
MOVL C01944 V=800.0 PL=0
MOVL C01945 V=800.0 PL=0
MOVL C01946 V=800.0 PL=0
MOVL C01947 V=800.0 PL=0
MOVL C01948 V=800.0 PL=0
MOVL C01949 V=800.0 PL=0
MOVL C01950 V=800.0 PL=0
MOVL C01951 V=800.0 PL=0
MOVL C01952 V=800.0 PL=0
MOVL C01953 V=800.0 PL=0
MOVL C01954 V=800.0 PL=0
MOVL C01955 V=800.0 PL=0
MOVL C01956 V=800.0 PL=0
MOVL C01957 V=800.0 PL=0
MOVL C01958 V=800.0 PL=0
MOVL C01959 V=800.0 PL=0
MOVL C01960 V=800.0 PL=0
MOVL C01961 V=800.0 PL=0
MOVL C01962 V=800.0 PL=0
MOVL C01963 V=800.0 PL=0
MOVL C01964 V=800.0 PL=0
MOVL C01965 V=800.0 PL=0
MOVL C01966 V=800.0 PL=0
MOVL C01967 V=800.0 PL=0
MOVL C01968 V=800.0 PL=0
MOVL C01969 V=800.0 PL=0
MOVL C01970 V=800.0 PL=0
MOVL C01971 V=800.0 PL=0
MOVL C01972 V=800.0 PL=0
MOVL C01973 V=800.0 PL=0
MOVL C01974 V=800.0 PL=0
MOVL C01975 V=800.0 PL=0
MOVL C01976 V=800.0 PL=0
MOVL C01977 V=800.0 PL=0
MOVL C01978 V=800.0 PL=0
MOVL C01979 V=800.0 PL=0
MOVL C01980 V=800.0 PL=0
MOVL C01981 V=800.0 PL=0
MOVL C01982 V=800.0 PL=0
MOVL C01983 V=800.0 PL=0
MOVL C01984 V=800.0 PL=0
MOVL C01985 V=800.0 PL=0
MOVL C01986 V=800.0 PL=0
MOVL C01987 V=800.0 PL=0
MOVL C01988 V=800.0 PL=0
MOVL C01989 V=800.0 PL=0
MOVL C01990 V=800.0 PL=0
MOVL C01991 V=800.0 PL=0
MOVL C01992 V=800.0 PL=0
MOVL C01993 V=800.0 PL=0
MOVL C01994 V=800.0 PL=0
MOVL C01995 V=800.0 PL=0
MOVL C01996 V=800.0 PL=0
MOVL C01997 V=800.0 PL=0
MOVL C01998 V=800.0 PL=0
MOVL C01999 V=800.0 PL=0
MOVL C02000 V=800.0 PL=0
MOVL C02001 V=800.0 PL=0
MOVL C02002 V=800.0 PL=0
MOVL C02003 V=800.0 PL=0
MOVL C02004 V=800.0 PL=0
MOVL C02005 V=800.0 PL=0
MOVL C02006 V=800.0 PL=0
MOVL C02007 V=800.0 PL=0
MOVL C02008 V=800.0 PL=0
MOVL C02009 V=800.0 PL=0
MOVL C02010 V=800.0 PL=0
MOVL C02011 V=800.0 PL=0
MOVL C02012 V=800.0 PL=0
MOVL C02013 V=800.0 PL=0
MOVL C02014 V=800.0 PL=0
MOVL C02015 V=800.0 PL=0
MOVL C02016 V=800.0 PL=0
MOVL C02017 V=800.0 PL=0
MOVL C02018 V=800.0 PL=0
MOVL C02019 V=800.0 PL=0
MOVL C02020 V=800.0 PL=0
MOVL C02021 V=800.0 PL=0
MOVL C02022 V=800.0 PL=0
MOVL C02023 V=800.0 PL=0
MOVL C02024 V=800.0 PL=0
MOVL C02025 V=800.0 PL=0
MOVL C02026 V=800.0 PL=0
MOVL C02027 V=800.0 PL=0
MOVL C02028 V=800.0 PL=0
MOVL C02029 V=800.0 PL=0
MOVL C02030 V=800.0 PL=0
MOVL C02031 V=800.0 PL=0
MOVL C02032 V=800.0 PL=0
MOVL C02033 V=800.0 PL=0
MOVL C02034 V=800.0 PL=0
MOVL C02035 V=800.0 PL=0
MOVL C02036 V=800.0 PL=0
MOVL C02037 V=800.0 PL=0
MOVL C02038 V=800.0 PL=0
MOVL C02039 V=800.0 PL=0
MOVL C02040 V=800.0 PL=0
MOVL C02041 V=800.0 PL=0
MOVL C02042 V=800.0 PL=0
MOVL C02043 V=800.0 PL=0
MOVL C02044 V=800.0 PL=0
MOVL C02045 V=800.0 PL=0
MOVL C02046 V=800.0 PL=0
MOVL C02047 V=800.0 PL=0
MOVL C02048 V=800.0 PL=0
MOVL C02049 V=800.0 PL=0
MOVL C02050 V=800.0 PL=0
MOVL C02051 V=800.0 PL=0
MOVL C02052 V=800.0 PL=0
MOVL C02053 V=800.0 PL=0
MOVL C02054 V=800.0 PL=0
MOVL C02055 V=800.0 PL=0
MOVL C02056 V=800.0 PL=0
MOVL C02057 V=800.0 PL=0
MOVL C02058 V=800.0 PL=0
MOVL C02059 V=800.0 PL=0
MOVL C02060 V=800.0 PL=0
MOVL C02061 V=800.0 PL=0
MOVL C02062 V=800.0 PL=0
MOVL C02063 V=800.0 PL=0
MOVL C02064 V=800.0 PL=0
MOVL C02065 V=800.0 PL=0
MOVL C02066 V=800.0 PL=0
MOVL C02067 V=800.0 PL=0
MOVL C02068 V=800.0 PL=0
MOVL C02069 V=800.0 PL=0
MOVL C02070 V=800.0 PL=0
MOVL C02071 V=800.0 PL=0
MOVL C02072 V=800.0 PL=0
MOVL C02073 V=800.0 PL=0
MOVL C02074 V=800.0 PL=0
MOVL C02075 V=800.0 PL=0
MOVL C02076 V=800.0 PL=0
MOVL C02077 V=800.0 PL=0
MOVL C02078 V=800.0 PL=0
MOVL C02079 V=800.0 PL=0
MOVL C02080 V=800.0 PL=0
MOVL C02081 V=800.0 PL=0
MOVL C02082 V=800.0 PL=0
MOVL C02083 V=800.0 PL=0
MOVL C02084 V=800.0 PL=0
MOVL C02085 V=800.0 PL=0
MOVL C02086 V=800.0 PL=0
MOVL C02087 V=800.0 PL=0
MOVL C02088 V=800.0 PL=0
MOVL C02089 V=800.0 PL=0
MOVL C02090 V=800.0 PL=0
MOVL C02091 V=800.0 PL=0
MOVL C02092 V=800.0 PL=0
MOVL C02093 V=800.0 PL=0
MOVL C02094 V=800.0 PL=0
MOVL C02095 V=800.0 PL=0
MOVL C02096 V=800.0 PL=0
MOVL C02097 V=800.0 PL=0
MOVL C02098 V=800.0 PL=0
MOVL C02099 V=800.0 PL=0
MOVL C02100 V=800.0 PL=0
MOVL C02101 V=800.0 PL=0
MOVL C02102 V=800.0 PL=0
MOVL C02103 V=800.0 PL=0
MOVL C02104 V=800.0 PL=0
MOVL C02105 V=800.0 PL=0
MOVL C02106 V=800.0 PL=0
MOVL C02107 V=800.0 PL=0
MOVL C02108 V=800.0 PL=0
MOVL C02109 V=800.0 PL=0
MOVL C02110 V=800.0 PL=0
MOVL C02111 V=800.0 PL=0
MOVL C02112 V=800.0 PL=0
MOVL C02113 V=800.0 PL=0
MOVL C02114 V=800.0 PL=0
MOVL C02115 V=800.0 PL=0
MOVL C02116 V=800.0 PL=0
MOVL C02117 V=800.0 PL=0
MOVL C02118 V=800.0 PL=0
MOVL C02119 V=800.0 PL=0
MOVL C02120 V=800.0 PL=0
MOVL C02121 V=800.0 PL=0
MOVL C02122 V=800.0 PL=0
MOVL C02123 V=800.0 PL=0
MOVL C02124 V=800.0 PL=0
